(* PLC project H2-1.0.02.project, CODESYS CODESYS V3.5 SP21 Patch 1 *)
(* stored: creationDateTime 2025-11-10T13:44:26.7492399, modificationDateTime 2025-11-05T06:53:28.9174298 *)

{attribute 'qualified_only'}
{attribute 'to_string'}
TYPE Duplex_Mapping : (Z100 := 0, Z201, Z202, TK201, Duplex_End);
END_TYPE

{attribute 'qualified_only'}
{attribute 'to_string'}
TYPE ME44DO_Mapping : (GW202_S4 := 0, GW201_S3, ME44DO_End);
END_TYPE

{attribute 'qualified_only'}
{attribute 'to_string'}
TYPE mPump_Mapping : (mPump_001 := 0, mPump_End);
END_TYPE

{attribute 'qualified_only'}
{attribute 'to_string'}
TYPE s8228_Mapping : (CT_122 := 0, CT_131, CT_142, s8228_End);
END_TYPE

{attribute 'qualified_only'}
{attribute 'to_string'}
TYPE DI_Mapping : (External_Pump_Status := 0, DC_OK, Z201_DC_OK, Spare_3, DI_End);
END_TYPE

{attribute 'qualified_only'}
{attribute 'to_string'}
TYPE Analog_Pump_Mapping : (Analog_Pump_001 := 0, Analog_Pump_End);
END_TYPE

(* values of LS_Mapping: LSLL_101: Z100; LSLL_202: Z201; LSHH_206: Z202-Filter 204A; LSHH_207: Z202-Filter 204B; LSHH_208: Z202-Filter 205A; LSHH_209: Z202-Filter 205B; LSHH_201: EP101; LSHH_204: TK201, *)

{attribute 'qualified_only'}
{attribute 'to_string'}
TYPE LS_Mapping : (LSLL_101 := 0, LSLL_202, LSHH_206, LSLL_210, LSHH_207, LSLL_211, LSHH_208, LSLL_212, LSHH_209, LSLL_213, LSHH_201, LSHH_204, LSLL_203, LSLL_205, LS_End);
END_TYPE

(* values of FIT_Mapping: FT01: FIT_111:=0, FIT_121, *)

{attribute 'qualified_only'}
{attribute 'to_string'}
TYPE FIT_Mapping : (FT01, FIT_End);
END_TYPE

{attribute 'qualified_only'}
{attribute 'to_string'}
TYPE Adam_6217_Mapping : (Adam_6217_001 := 0, Adam_6217_End);
END_TYPE

{attribute 'qualified_only'}
{attribute 'to_string'}
TYPE Adam_6250_Mapping : (Adam_6250_001 := 1, Adam_6250_002, Adam_End);
END_TYPE

(* values of s8098_Mapping: FT_101: Z100; FT_201: Z201; FT_202: Z202; FT_203: TK201 *)

{attribute 'qualified_only'}
{attribute 'to_string'}
TYPE s8098_Mapping : (FT_101 := 0, FT_201, FT_202, FT_204, FT_203, s8098_end);
END_TYPE

(* values of ME44AI_Mapping: GW201_S2: 2; GW201_S4: 4 *)

(* {attribute 'strict'} *)
{attribute 'qualified_only'}
{attribute 'to_string'}
TYPE ME44AI_Mapping : (GW100_S2 := 0, GW100_S3, GW201_S2, GW202_S3, GW201_S4, ME44_AI_End);
END_TYPE

(* values of VFD_Mapping: VFD_101A: VFD-101; VFD_201: Z201; VFD_202: Z202; VFD_102A: EP101; VFD_203: TK201 *)

{attribute 'qualified_only'}
{attribute 'to_string'}
TYPE VFD_Mapping : (VFD_101A := 0, VFD_101B, VFD_201, VFD_201B, VFD_202, VFD_202B, VFD_102A, VFD_102B, VFD_102C, VFD_102D, VFD_102E, VFD_102F, VFD_102G, VFD_102H, VFD_203, VFD_End);
END_TYPE

{attribute 'qualified_only'}
{attribute 'to_string'}
TYPE b8653_mapping : (enum_member := 0, b8653_End);
END_TYPE

(* values of BCV_Mapping: BCV_211: Z202-Filter 204A; BCV_212: Z202-Filter 204B; BCV_217: Z202-Filter 205A; BCV_218: Z202-Filter 205B *)

{attribute 'qualified_only'}
{attribute 'to_string'}
TYPE BCV_Mapping : (BCV_211, BCV_220, BCV_212, BCV_221, BCV_217, BCV_222, BCV_218, BCV_223, BCV_END);
END_TYPE

{attribute 'qualified_only'}
{attribute 'to_string'}
TYPE me64_Mapping : (ME64_001 := 0, ME64_End);
END_TYPE

(* values of Do_Mapping: Stack_R: 5; Skid_201_PWR: 9 *)

{attribute 'qualified_only'}
{attribute 'to_string'}
TYPE Do_Mapping : (Filters_204A := 0, Filters_204B, Filters_205A, Filters_205B, FilterSkid, Stack_R, Stack_Y, Stack_G, Stack_H, Skid_201_PWR, Skid_203_PWR, TK201_PWR_1, TK201_PWR_2, TK201_PWR_3, Do_End);
END_TYPE

(* 8312 Temperature *)
{attribute 'qualified_only'}
{attribute 'to_string'}
TYPE s8412_Mapping : (s8412_001 := 0, s8412_End);
END_TYPE

(* values of s3363_Mapping: ACV_101: Z100; ACV_201: Z201; ACV_207: 3; ACV_208: 5; ACV_213: 7; ACV_214: 9; ACV_219: Z202; ACV_203: TK201 *)

(* {attribute 'strict'} *)
{attribute 'qualified_only'}
{attribute 'to_string'}
TYPE s3363_Mapping : (ACV_101 := 0, ACV_102, ACV_201, ACV_207, ACV_209, ACV_208, ACV_210, ACV_213, ACV_215, ACV_214, ACV_216, ACV_219, ACV_203, ACV_206, ACV_224, ACV_225, ACV_226, s3363_END);
END_TYPE

(* values of s8312_Mapping: PT_101: Z100; PT_201: Z201; PT_202: Z202; PT_203: TK201 *)

(* 8312 Pressure *)
{attribute 'qualified_only'}
{attribute 'to_string'}
TYPE s8312_Mapping : (PT_101 := 0, PT_201, PT_202, PT_204, PT_205, PT_203, S8312_End);
END_TYPE

{attribute 'qualified_only'}
{attribute 'to_string'}
TYPE ME44AO_Mapping : (ME44AO := 0, ME44AO_End);
END_TYPE

{attribute 'qualified_only'}
{attribute 'to_string'}
TYPE Stack_Light_Mapping : (Stack_Light_001 := 0, Stack_Light_End);
END_TYPE

(* values of Line_Mapping: Line_End: Line_3, Line_4, *)

{attribute 'qualified_only'}
{attribute 'to_string'}
TYPE Line_Mapping : (Water := 0, Bleach, Line_End);
END_TYPE

(* values of s8050_Mapping: FT_201A: Z201; FT_202A: Z202; FT_203A: TK201 *)

{attribute 'qualified_only'}
{attribute 'to_string'}
TYPE s8050_Mapping : (FT_201A := 0, FT_202A, FT_204A, FT_203A, s8050_End);
END_TYPE

{attribute 'qualified_only'}
{attribute 'to_string'}
TYPE TT_Mapping : (TT_Start := 0, TT_End);
END_TYPE

(* values of PID_Mapping: Z201_EP101_Level: 3; Z202_Flow: 6; Z202_TK201_Level: 8; TK201_Flow: 11 *)

{attribute 'qualified_only'}
{attribute 'to_string'}
TYPE PID_Mapping : (Z100_Flow := 0, Z100_Pressure, Z100_Level, Z201_EP101_Level, Z201_TK201_Level, Z201_Flow, Z202_Flow, Z202_Pressure, Z202_TK201_Level, Z202_EP101_Level, Z202_Filter_Flow, TK201_Flow, TK201_Pressure, Z202_Recovery_Level, PID_End);
END_TYPE

{attribute 'qualified_only'}
{attribute 'to_string'}
TYPE SV_Mapping : (SV_001 := 0, SV_END);
END_TYPE

(* values of AIT_Mapping: LT_101_P: EP101; LT_202: TK201; LT_202A: 5; LT_01A: 7 *)

{attribute 'qualified_only'}
{attribute 'to_string'}
TYPE AIT_Mapping : (LT_101_P := 0, LT_101_T, LT_201, LT_201A_P, LT_201A_T, LT_202, LT_202A, LT_01A, LT_01B, FT_01, UV_001, AIT_End);
END_TYPE

{attribute 'qualified_only'}
{attribute 'to_string'}
TYPE ACV_Mapping : (ACV_111 := 0, ACV_121, ACV_End);
END_TYPE

(* values of s8605_Mapping: SV_211: Z202-Filter 204A; SV_212: Z202-Filter 204B; SV_217: Z202-Filter 205A; SV_218: Z202-Filter 204A *)

{attribute 'qualified_only'}
{attribute 'to_string'}
TYPE s8605_Mapping : (SV_211 := 0, SV_220, SV_212, SV_221, SV_217, SV_222, SV_218, SV_223, s8605_End);
END_TYPE

{attribute 'qualified_only'}
{attribute 'to_string'}
TYPE ME44DI_Mapping : (GW100_S1 := 0, GW201_S1, GW202_S1, GW202_S2, Me44DI_End);
END_TYPE

PROGRAM Z201_Manager
  VAR
    Local_Status : eZ201_Status;
    tStatus : eZ201_Status;
    Local_Task : eZ201_Task;
    tAlarm : Burkert.Alarm_Window;
    LT201_tAlarm : Burkert.Alarm_Window;
    FT201_Ave : REAL;
    FT201_Gav : REAL;
    FT201_Hav : REAL;
    FT201_Ave_Index : INT;
    Array_Size : UINT;
    VFD_Min_PCT : REAL := 20;
    Level_ton : ton;
  END_VAR
  VAR  (* added by the conversion: wires and edge detectors of the diagram *)
    _SEL3_OUT : ANY;
    _SEL3_OUT_2 : ANY;
    _OR5_OUT : BOOL;
    _SEL21_OUT : ANY;
    _SEL35_OUT : ANY;
    _MAX51_OUT : ANY;
    _LIMIT47_OUT : REAL;
    _GT62_OUT : BOOL;
    _SEL75_OUT : REAL;
    _GT86_OUT : BOOL;
  END_VAR

            PVL.Z201_Config.Mode.eMode:=Burkert.eHOA_Modes.Manual;

Aux();
Alarms();

PVL.Z201_Config.StrMode:=Burkert.Burkert_OSCAT_BASIC.REPLACE_ALL(str:=TO_STRING(PVL.Z201_Config.Mode.eMode) , src:='_' , rep:=' ' );
PVL.Z201_Config.StrStatus:=Burkert.Burkert_OSCAT_BASIC.REPLACE_ALL(str:=TO_STRING(PVL.Z201_Config.Status.eStatus) , src:='_' , rep:=' ' );
PVl.Z201_Config.StrTask:=Burkert.Burkert_OSCAT_BASIC.REPLACE_ALL(str:=TO_STRING(PVL.Z201_Config.Task.eTask) , src:='_' , rep:=' ' );




CASE PVL.Z201_Config.Mode.eMode OF
	Burkert.eHOA_Modes.Off:PVL.Z201_Config.Task.eTask:=eZ201_task.Off;
	//Burkert.eHOA_Modes.Auto:
	//Burkert.eHOA_Modes.Manual:
END_CASE;

CASE pvl.Z201_Config.Task.eTask OF
	eZ201_Task.Off:Task_Off();
	eZ201_Task.Flow:Task_Flow();
	eZ201_Task.TK201_Level:TK201_level();
	eZ201_task.EP101_Level:EP101_Level();
	eZ201_Task.Z100_Flow:Z100_Flow();
	eZ201_Task.Z202_Flow:Z202_Flow();
	eZ201_Task.Drain:Drain();	
	eZ201_Task.Agitate_only:Task_Agitate();
END_CASE





PID_ctrl();
ACV_ctrl();
VFD_ctrl();



          

ACTION Task_Flow:
                IF PVL.Z201_Config.Task.eTask<> Local_Task THEN
	Local_Task:=PVL.Z201_Config.Task.eTask;
	Local_Status:=eZ201_Status.Fixed_Flow_Rate_Transfer_Active;
END_IF;






PVL.PID[PID_Mapping.Z201_Flow].PLC_Target:=PVL.Z201_Config.Target_Flow.Target;


	
	


CASE PVL.Z201_Config.Status.eStatus OF
	
	eZ201_Status.PT201_High_Pressure_Alarm:		Local_Status:=PVL.Z201_Config.Status.eStatus;
	eZ201_Status.PT201_Low_Pressure_Alarm:		Local_Status:=PVL.Z201_Config.Status.eStatus;
	eZ201_Status.FT201_Low_Low_Flow_Alarm:		Local_Status:=PVL.Z201_Config.Status.eStatus;
	//eZ201_Status.LT101_High_High_Alarm:			Local_Status:=PVL.Z201_Config.Status.eStatus;
	//eZ201_Status.LT101_Low_Low_Alarm:			Local_Status:=PVL.Z201_Config.Status.eStatus;
	//eZ201_Status.LT201_High_High_Alarm:			Local_Status:=PVL.Z201_Config.Status.eStatus;
	//eZ201_Status.LT201_Low_Low_Alarm:			Local_Status:=PVL.Z201_Config.Status.eStatus;
	//eZ201_Status.LT201A_High_High_Alarm:		Local_Status:=PVL.Z201_Config.Status.eStatus;
	//eZ201_Status.LT201A_Low_Low_Alarm:			Local_Status:=PVL.Z201_Config.Status.eStatus;
	eZ201_Status.TK201_LSHH204_High_High_Level_Alarm:	Local_Status:=PVL.Z201_Config.Status.eStatus;
	eZ201_Status.Pump_Intake_Dry_LSLL202:		Local_Status:=PVL.Z201_Config.Status.eStatus;
	//eZ201_Status.PT201_High_Pressure_Alarm:		Local_Status:=PVL.Z201_Config.Status.eStatus;
	///eZ201_Status.PT201_Low_Pressure_Alarm:		Local_Status:=PVL.Z201_Config.Status.eStatus;
	//eZ201_Status.FT201_Low_Low_Flow_Alarm:		Local_Status:=PVL.Z201_Config.Status.eStatus;
	
	eZ201_Status.LT201_Low_Low_Alarm:		IF Level_ton.Q THEN local_Status:= eZ201_Status.Waiting_For_Level_OK_LT201; END_IF;
	eZ201_Status.LT202_High_High_Alarm:		IF Level_ton.Q THEN local_Status:= eZ201_Status.Waiting_For_Level_OK_LT202; END_IF;
	eZ201_Status.Waiting_For_Level_OK_LT201:	IF PVL.AIT[AIT_Mapping.LT_201].Status.eStatus=Burkert.eSensor_Status.OK THEN Local_Task:=999; END_IF;
	eZ201_Status.Waiting_For_Level_OK_LT202:	IF PVL.AIT[AIT_Mapping.LT_202].Status.eStatus=Burkert.eSensor_Status.OK THEN Local_Task:=999; END_IF;
	
	eZ201_Status.LT202A_High_High_Alarm:			Local_Status:=eZ201_Status.Waiting_For_Level_OK_LT202a;
	eZ201_Status.Waiting_For_Level_OK_LT202a	:	IF PVL.AIT[ait_mapping.LT_101_P].Status.eStatus=Burkert.eSensor_Status.OK THEN local_Task:=99; END_IF;
	
	

END_CASE;

Evaluate_Task_Flow();
              
END_ACTION

ACTION Z202_Flow:
                IF PVL.Z201_Config.Task.eTask<> Local_Task THEN
	Local_Task:=PVL.Z201_Config.Task.eTask;
END_IF;

Local_Status:=eZ201_Status.Z202_Rate_Match_Transfer_Active;




PVL.PID[PID_Mapping.Z201_Flow].PLC_Target:=PVL.s8098[s8098_Mapping.FT_203].PDO.VolumeFlow.EU;



Evaluate_Z202_Flow();

CASE PVL.Z201_Config.Status.eStatus OF
	//eZ201_Status.LT101_High_High_Alarm:			Local_Status:=PVL.Z201_Config.Status.eStatus;
	//eZ201_Status.LT101_Low_Low_Alarm:			Local_Status:=PVL.Z201_Config.Status.eStatus;
	//eZ201_Status.LT201_High_High_Alarm:			Local_Status:=PVL.Z201_Config.Status.eStatus;
	//eZ201_Status.LT201_Low_Low_Alarm:			Local_Status:=PVL.Z201_Config.Status.eStatus;
	//eZ201_Status.LT201A_High_High_Alarm:		Local_Status:=PVL.Z201_Config.Status.eStatus;
	//eZ201_Status.LT201A_Low_Low_Alarm:			Local_Status:=PVL.Z201_Config.Status.eStatus;
	eZ201_Status.TK201_LSHH204_High_High_Level_Alarm:	Local_Status:=PVL.Z201_Config.Status.eStatus;
	eZ201_Status.Pump_Intake_Dry_LSLL202:		Local_Status:=PVL.Z201_Config.Status.eStatus;
	eZ201_Status.PT201_High_Pressure_Alarm:		Local_Status:=PVL.Z201_Config.Status.eStatus;
	///eZ201_Status.PT201_Low_Pressure_Alarm:		Local_Status:=PVL.Z201_Config.Status.eStatus;
	eZ201_Status.FT201_Low_Low_Flow_Alarm:		Local_Status:=PVL.Z201_Config.Status.eStatus;
	eZ201_Status.LT201_Low_Low_Alarm:		IF Level_ton.Q THEN local_Status:= eZ201_Status.Waiting_For_Level_OK_LT201; END_IF;
	eZ201_Status.LT202_High_High_Alarm:		IF Level_ton.Q THEN local_Status:= eZ201_Status.Waiting_For_Level_OK_LT202; END_IF;
	eZ201_Status.Waiting_For_Level_OK_LT201:	IF PVL.AIT[AIT_Mapping.LT_201].Status.eStatus=Burkert.eSensor_Status.OK THEN Local_Task:=999; END_IF;
	eZ201_Status.Waiting_For_Level_OK_LT202:	IF PVL.AIT[AIT_Mapping.LT_202].Status.eStatus=Burkert.eSensor_Status.OK THEN Local_Task:=999; END_IF;
	eZ201_Status.LT202A_High_High_Alarm:			Local_Status:=eZ201_Status.Waiting_For_Level_OK_LT202a;
	eZ201_Status.Waiting_For_Level_OK_LT202a	:	IF PVL.AIT[ait_mapping.LT_101_P].Status.eStatus=Burkert.eSensor_Status.OK THEN local_Task:=99; END_IF;
	

	eZ201_Status.PT201_Low_Pressure_Alarm:		Local_Status:=PVL.Z201_Config.Status.eStatus;
	//eZ201_Status.FT201_Low_Low_Flow_Alarm:		Local_Status:=PVL.Z201_Config.Status.eStatus;

END_CASE
              
END_ACTION

ACTION Task_OFF:
                IF PVL.Z201_Config.Task.eTask<> Local_Task THEN
	Local_Task:=PVL.Z201_Config.Task.eTask;
END_IF;

Local_Status:=eZ201_Status.Off;

Evaluate_Off();

              
END_ACTION

ACTION Drain:
                IF PVL.Z201_Config.Task.eTask<> Local_Task THEN
	Local_Task:=PVL.Z201_Config.Task.eTask;
	Local_Status:=eZ201_Status.Drain_Active;
END_IF;






PVL.PID[PID_Mapping.Z201_Flow].PLC_Target:=PVl.Z201_Config.Drain_Rate.Target;



Evaluate_Drain();


CASE PVL.Z201_Config.Status.eStatus OF
	//eZ201_Status.LT101_High_High_Alarm:			Local_Status:=PVL.Z201_Config.Status.eStatus;
	//eZ201_Status.LT101_Low_Low_Alarm:			Local_Status:=PVL.Z201_Config.Status.eStatus;
	//eZ201_Status.LT201_High_High_Alarm:			Local_Status:=PVL.Z201_Config.Status.eStatus;
	//eZ201_Status.LT201_Low_Low_Alarm:			Local_Status:=PVL.Z201_Config.Status.eStatus;
	//eZ201_Status.LT201A_High_High_Alarm:		Local_Status:=PVL.Z201_Config.Status.eStatus;
	//eZ201_Status.LT201A_Low_Low_Alarm:			Local_Status:=PVL.Z201_Config.Status.eStatus;
	//eZ201_Status.TK201_High_High_Level_Alarm:	Local_Status:=PVL.Z201_Config.Status.eStatus;
	eZ201_Status.Pump_Intake_Dry_LSLL202:		Local_Status:=PVL.Z201_Config.Status.eStatus;
	eZ201_Status.Drain_Complete:				Local_Status:=PVL.Z201_Config.Status.eStatus;
	
	eZ201_Status.PT201_High_Pressure_Alarm:		Local_Status:=eZ201_Status.PT201_High_Pressure_Alarm;
	eZ201_Status.PT201_Low_Pressure_Alarm:		Local_Status:=eZ201_Status.PT201_Low_Pressure_Alarm;
	eZ201_Status.FT201_Low_Low_Flow_Alarm:		Local_Status:=eZ201_Status.FT201_Low_Low_Flow_Alarm;
	
	eZ201_Status.LT201_Low_Low_Alarm:		IF Level_ton.Q THEN local_Status:= eZ201_Status.Waiting_For_Level_OK_LT201; END_IF;
	eZ201_Status.LT202_High_High_Alarm:		IF Level_ton.Q THEN local_Status:= eZ201_Status.Waiting_For_Level_OK_LT202; END_IF;
	eZ201_Status.Waiting_For_Level_OK_LT201:	IF PVL.AIT[AIT_Mapping.LT_201].Status.eStatus=Burkert.eSensor_Status.OK THEN Local_Task:=999; END_IF;
	eZ201_Status.Waiting_For_Level_OK_LT202:	IF PVL.AIT[AIT_Mapping.LT_202].Status.eStatus=Burkert.eSensor_Status.OK THEN Local_Task:=999; END_IF;
	
	eZ201_Status.LT202A_High_High_Alarm:			Local_Status:=eZ201_Status.Waiting_For_Level_OK_LT202a;
	eZ201_Status.Waiting_For_Level_OK_LT202a	:	IF PVL.AIT[ait_mapping.LT_101_P].Status.eStatus=Burkert.eSensor_Status.OK THEN local_Task:=99; END_IF;
	

END_CASE;
              
END_ACTION

ACTION Evaluate_Off:
                tStatus:=Local_Status;

IF GVl.LS[LS_Mapping.LSLL_202].Status.eStatus=Burkert.DI_Status.No_Liquid_Detected_Alarm THEN tStatus:=eZ201_Status.Pump_Intake_Dry_LSLL202; END_IF;
IF GVl.LS[LS_Mapping.LSHH_204 ].Status.eStatus=Burkert.DI_Status.Liquid_Detected_Alarm THEN tStatus:=eZ201_Status.TK201_LSHH204_High_High_Level_Alarm; END_IF;

//IF NOT(Network.VFD[VFD_Mapping.VFD_102A].Ready) THEN tStatus:=eZ201_Status.VFD_102A_Not_Ready;	END_IF;
//IF NOT(Network.VFD[VFD_Mapping.VFD_102B].Ready) THEN tStatus:=eZ201_Status.VFD_102B_Not_Ready;	END_IF;
//IF NOT(Network.VFD[VFD_Mapping.VFD_102C].Ready) THEN tStatus:=eZ201_Status.VFD_102C_Not_Ready;	END_IF;
//IF NOT(Network.VFD[VFD_Mapping.VFD_102D].Ready) THEN tStatus:=eZ201_Status.VFD_102D_Not_Ready;	END_IF;
//IF NOT(Network.VFD[VFD_Mapping.VFD_102E].Ready) THEN tStatus:=eZ201_Status.VFD_102E_Not_Ready;	END_IF;
//IF NOT(Network.VFD[VFD_Mapping.VFD_102F].Ready) THEN tStatus:=eZ201_Status.VFD_102F_Not_Ready;	END_IF;
//IF NOT(Network.VFD[VFD_Mapping.VFD_102G].Ready) THEN tStatus:=eZ201_Status.VFD_102G_Not_Ready;	END_IF;
//IF NOT(Network.VFD[VFD_Mapping.VFD_102H].Ready) THEN tStatus:=eZ201_Status.VFD_102H_Not_Ready;	END_IF;

IF Network.VFD[VFD_Mapping.VFD_102A].Status=Burkert.eVFD_Status.High_High_Current_Alarm THEN tStatus:=eZ201_Status.VFD_102A_High_Current;	END_IF;
IF Network.VFD[VFD_Mapping.VFD_102B].Status=Burkert.eVFD_Status.High_High_Current_Alarm THEN tStatus:=eZ201_Status.VFD_102B_High_Current;	END_IF;
IF Network.VFD[VFD_Mapping.VFD_102C].Status=Burkert.eVFD_Status.High_High_Current_Alarm THEN tStatus:=eZ201_Status.VFD_102C_High_Current;	END_IF;
IF Network.VFD[VFD_Mapping.VFD_102D].Status=Burkert.eVFD_Status.High_High_Current_Alarm THEN tStatus:=eZ201_Status.VFD_102D_High_Current;	END_IF;
//IF Network.VFD[VFD_Mapping.VFD_102E].Status=Burkert.eVFD_Status.High_High_Current_Alarm THEN tStatus:=eZ201_Status.VFD_102E_High_Current;	END_IF;
//IF Network.VFD[VFD_Mapping.VFD_102F].Status=Burkert.eVFD_Status.High_High_Current_Alarm THEN tStatus:=eZ201_Status.VFD_102F_High_Current;	END_IF;
//IF Network.VFD[VFD_Mapping.VFD_102G].Status=Burkert.eVFD_Status.High_High_Current_Alarm THEN tStatus:=eZ201_Status.VFD_102G_High_Current;	END_IF;
//IF Network.VFD[VFD_Mapping.VFD_102H].Status=Burkert.eVFD_Status.High_High_Current_Alarm THEN tStatus:=eZ201_Status.VFD_102H_High_Current;	END_IF;


IF NOT(Network.VFD[VFD_Mapping.VFD_201].Ready) THEN tStatus:=eZ201_Status.VFD_201_Not_Ready;	END_IF;

IF NOT(GVL.s3363[s3363_mapping.ACV_201].Ready) THEN	tStatus:=eZ201_Status.ACV_201_Not_Ready;	END_IF;
	
IF NOT(PVl.s8312[s8312_mapping.PT_201].Ready) THEN	tStatus:=eZ201_status.PT201_Not_Ready;	END_IF;
IF NOT(PVL.s8098[s8098_Mapping.FT_201].Ready) THEN	tStatus:=eZ201_status.FT201_Not_Ready;	END_IF;


IF NOT(PVL.AIT[AIT_Mapping.LT_101_P].Ready) THEN tStatus:=eZ201_Status.LT101_Not_Ready;	END_IF;
IF NOT(PVL.AIT[AIT_Mapping.LT_201A_P].Ready) THEN tStatus:=eZ201_Status.LT201A_Not_Ready;	END_IF;
IF NOT(PVL.AIT[AIT_Mapping.LT_201].Ready) THEN tStatus:=eZ201_Status.LT201_Not_Ready;	END_IF;

IF PVL.AIT[AIT_Mapping.LT_101_P].Status.eStatus=Burkert.eSensor_Status.HiHi_Alarm THEN	tStatus:=eZ201_Status.LT101_High_High_Alarm; END_IF;
IF PVL.AIT[AIT_Mapping.LT_101_P].Status.eStatus=Burkert.eSensor_Status.Low_Low_Alarm THEN	tStatus:=eZ201_Status.LT101_Low_Low_Alarm; END_IF;

IF PVL.AIT[AIT_Mapping.LT_201A_P].Status.eStatus=Burkert.eSensor_Status.HiHi_Alarm THEN	tStatus:=eZ201_Status.LT201A_High_High_Alarm; END_IF;
IF PVL.AIT[AIT_Mapping.LT_201A_P].Status.eStatus=Burkert.eSensor_Status.Low_Low_Alarm THEN	tStatus:=eZ201_Status.LT201A_Low_Low_Alarm; END_IF;

IF PVL.AIT[AIT_Mapping.LT_201].Status.eStatus=Burkert.eSensor_Status.HiHi_Alarm THEN	tStatus:=eZ201_Status.LT201_High_High_Alarm; END_IF;
IF PVL.AIT[AIT_Mapping.LT_201].Status.eStatus=Burkert.eSensor_Status.Low_Low_Alarm THEN	tStatus:=eZ201_Status.LT201_Low_Low_Alarm; END_IF;


PVL.Z201_Config.Status.eStatus:=tStatus;

              
END_ACTION

ACTION Z100_Flow:
                IF PVL.Z201_Config.Task.eTask<> Local_Task THEN
	Local_Task:=PVL.Z201_Config.Task.eTask;
END_IF;

Local_Status:=eZ201_Status.Z100_Rate_Match_Transfer_Active;




PVL.PID[PID_Mapping.Z201_Flow].PLC_Target:=PVL.s8098[s8098_Mapping.FT_101].PDO.VolumeFlow.EU;




Evaluate_Z100_Flow();

CASE PVL.Z201_Config.Status.eStatus OF
	//eZ201_Status.LT101_High_High_Alarm:			Local_Status:=PVL.Z201_Config.Status.eStatus;
	//eZ201_Status.LT101_Low_Low_Alarm:			Local_Status:=PVL.Z201_Config.Status.eStatus;
	//eZ201_Status.LT201_High_High_Alarm:			Local_Status:=PVL.Z201_Config.Status.eStatus;
	//eZ201_Status.LT201_Low_Low_Alarm:			Local_Status:=PVL.Z201_Config.Status.eStatus;
	//eZ201_Status.LT201A_High_High_Alarm:		Local_Status:=PVL.Z201_Config.Status.eStatus;
	//eZ201_Status.LT201A_Low_Low_Alarm:			Local_Status:=PVL.Z201_Config.Status.eStatus;
	eZ201_Status.TK201_LSHH204_High_High_Level_Alarm:	Local_Status:=PVL.Z201_Config.Status.eStatus;
	eZ201_Status.Pump_Intake_Dry_LSLL202:		Local_Status:=PVL.Z201_Config.Status.eStatus;
	eZ201_Status.PT201_High_Pressure_Alarm:		Local_Status:=PVL.Z201_Config.Status.eStatus;
	///eZ201_Status.PT201_Low_Pressure_Alarm:		Local_Status:=PVL.Z201_Config.Status.eStatus;
	eZ201_Status.FT201_Low_Low_Flow_Alarm:		Local_Status:=PVL.Z201_Config.Status.eStatus;
	
	eZ201_Status.LT201_Low_Low_Alarm:		IF Level_ton.Q THEN local_Status:= eZ201_Status.Waiting_For_Level_OK_LT201; END_IF;
	eZ201_Status.LT202_High_High_Alarm:		IF Level_ton.Q THEN local_Status:= eZ201_Status.Waiting_For_Level_OK_LT202; END_IF;
	eZ201_Status.Waiting_For_Level_OK_LT201:	IF PVL.AIT[AIT_Mapping.LT_201].Status.eStatus=Burkert.eSensor_Status.OK THEN Local_Task:=999; END_IF;
	eZ201_Status.Waiting_For_Level_OK_LT202:	IF PVL.AIT[AIT_Mapping.LT_202].Status.eStatus=Burkert.eSensor_Status.OK THEN Local_Task:=999; END_IF;
	eZ201_Status.LT202A_High_High_Alarm:			Local_Status:=eZ201_Status.Waiting_For_Level_OK_LT202a;
	eZ201_Status.Waiting_For_Level_OK_LT202a	:	IF PVL.AIT[ait_mapping.LT_101_P].Status.eStatus=Burkert.eSensor_Status.OK THEN local_Task:=99; END_IF;
	
	//eZ201_Status.PT201_High_Pressure_Alarm:		Local_Status:=PVL.Z201_Config.Status.eStatus;
	eZ201_Status.PT201_Low_Pressure_Alarm:		Local_Status:=PVL.Z201_Config.Status.eStatus;
	//eZ201_Status.FT201_Low_Low_Flow_Alarm:		Local_Status:=PVL.Z201_Config.Status.eStatus;

END_CASE
              
END_ACTION

ACTION ACV_ctrl:
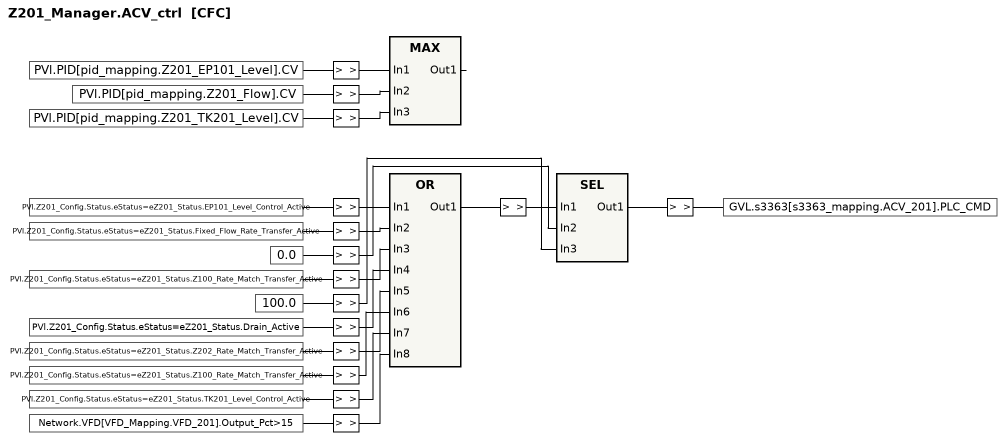
(* CFC diagram, written out as Structured Text *)
GVL.s3363[s3363_mapping.ACV_201].PLC_CMD := _SEL3_OUT;
_SEL3_OUT := SEL((PVl.Z201_Config.Status.eStatus=eZ201_Status.EP101_Level_Control_Active) OR (PVl.Z201_Config.Status.eStatus=eZ201_Status.Fixed_Flow_Rate_Transfer_Active) OR (PVl.Z201_Config.Status.eStatus=eZ201_Status.Z100_Rate_Match_Transfer_Active) OR (PVl.Z201_Config.Status.eStatus=eZ201_Status.Drain_Active) OR (PVl.Z201_Config.Status.eStatus=eZ201_Status.Z202_Rate_Match_Transfer_Active) OR (PVl.Z201_Config.Status.eStatus=eZ201_Status.Z100_Rate_Match_Transfer_Active) OR (PVl.Z201_Config.Status.eStatus=eZ201_Status.TK201_Level_Control_Active) OR (Network.VFD[VFD_Mapping.VFD_201].Output_Pct>15), 0.0, 100.0);
MAX(PVl.PID[pid_mapping.Z201_EP101_Level].CV, PVl.PID[pid_mapping.Z201_Flow].CV, PVl.PID[pid_mapping.Z201_TK201_Level].CV);
END_ACTION

ACTION Evaluate_Z100_Flow:
                tStatus:=Local_Status;

IF GVl.LS[LS_Mapping.LSLL_202].Status.eStatus=Burkert.DI_Status.No_Liquid_Detected_Alarm THEN tStatus:=eZ201_Status.Pump_Intake_Dry_LSLL202; END_IF;
IF GVl.LS[LS_Mapping.LSHH_204 ].Status.eStatus=Burkert.DI_Status.Liquid_Detected_Alarm THEN tStatus:=eZ201_Status.TK201_LSHH204_High_High_Level_Alarm; END_IF;

//IF NOT(Network.VFD[VFD_Mapping.VFD_102A].Ready) THEN tStatus:=eZ201_Status.VFD_102A_Not_Ready;	END_IF;
//IF NOT(Network.VFD[VFD_Mapping.VFD_102B].Ready) THEN tStatus:=eZ201_Status.VFD_102B_Not_Ready;	END_IF;
//IF NOT(Network.VFD[VFD_Mapping.VFD_102C].Ready) THEN tStatus:=eZ201_Status.VFD_102C_Not_Ready;	END_IF;
//IF NOT(Network.VFD[VFD_Mapping.VFD_102D].Ready) THEN tStatus:=eZ201_Status.VFD_102D_Not_Ready;	END_IF;
//IF NOT(Network.VFD[VFD_Mapping.VFD_102E].Ready) THEN tStatus:=eZ201_Status.VFD_102E_Not_Ready;	END_IF;
//IF NOT(Network.VFD[VFD_Mapping.VFD_102F].Ready) THEN tStatus:=eZ201_Status.VFD_102F_Not_Ready;	END_IF;
//IF NOT(Network.VFD[VFD_Mapping.VFD_102G].Ready) THEN tStatus:=eZ201_Status.VFD_102G_Not_Ready;	END_IF;
//IF NOT(Network.VFD[VFD_Mapping.VFD_102H].Ready) THEN tStatus:=eZ201_Status.VFD_102H_Not_Ready;	END_IF;
IF NOT(Network.VFD[VFD_Mapping.VFD_201].Ready) THEN tStatus:=eZ201_Status.VFD_201_Not_Ready;	END_IF;

//IF Network.VFD[VFD_Mapping.VFD_102A].Status=Burkert.eVFD_Status.High_High_Current_Alarm THEN tStatus:=eZ201_Status.VFD_102A_High_Current;	END_IF;
//IF Network.VFD[VFD_Mapping.VFD_102B].Status=Burkert.eVFD_Status.High_High_Current_Alarm THEN tStatus:=eZ201_Status.VFD_102B_High_Current;	END_IF;
//IF Network.VFD[VFD_Mapping.VFD_102C].Status=Burkert.eVFD_Status.High_High_Current_Alarm THEN tStatus:=eZ201_Status.VFD_102C_High_Current;	END_IF;
//IF Network.VFD[VFD_Mapping.VFD_102D].Status=Burkert.eVFD_Status.High_High_Current_Alarm THEN tStatus:=eZ201_Status.VFD_102D_High_Current;	END_IF;
//IF Network.VFD[VFD_Mapping.VFD_102E].Status=Burkert.eVFD_Status.High_High_Current_Alarm THEN tStatus:=eZ201_Status.VFD_102E_High_Current;	END_IF;
//IF Network.VFD[VFD_Mapping.VFD_102F].Status=Burkert.eVFD_Status.High_High_Current_Alarm THEN tStatus:=eZ201_Status.VFD_102F_High_Current;	END_IF;
//IF Network.VFD[VFD_Mapping.VFD_102G].Status=Burkert.eVFD_Status.High_High_Current_Alarm THEN tStatus:=eZ201_Status.VFD_102G_High_Current;	END_IF;
//IF Network.VFD[VFD_Mapping.VFD_102H].Status=Burkert.eVFD_Status.High_High_Current_Alarm THEN tStatus:=eZ201_Status.VFD_102H_High_Current;	END_IF;



IF NOT(GVL.s3363[s3363_mapping.ACV_201].Ready) THEN	tStatus:=eZ201_Status.ACV_201_Not_Ready;	END_IF;
	
IF NOT(PVl.s8312[s8312_mapping.PT_201].Ready) THEN	tStatus:=eZ201_status.PT201_Not_Ready;	END_IF;
IF PVL.s8312[s8312_Mapping.PT_201].Status.eStatus=Burkert.eSensor_Status.HiHi_Alarm THEN tStatus:=eZ201_Status.PT201_High_Pressure_Alarm; END_IF;
//IF PVL.s8312[s8312_Mapping.PT_201].Status.eStatus=Burkert.eSensor_Status.Low_Low_Alarm THEN tStatus:=eZ201_Status.PT201_Low_Pressure_Alarm; END_IF;

IF NOT(PVL.s8098[s8098_Mapping.FT_201].Ready) THEN	tStatus:=eZ201_status.FT201_Not_Ready;	END_IF;
IF PVL.s8098[s8098_Mapping.FT_201].PDO.VolumeFlow.Status.eStatus=Burkert.eSensor_Status.Low_Low_Alarm THEN tStatus:=eZ201_status.FT201_Low_Low_Flow_Alarm;	END_IF;


//IF NOT(PVL.AIT[AIT_Mapping.LT_101_P].Ready) THEN tStatus:=eZ201_Status.LT101_Not_Ready;	END_IF;
//IF NOT(PVL.AIT[AIT_Mapping.LT_201A_P].Ready) THEN tStatus:=eZ201_Status.LT201A_Not_Ready;	END_IF;
IF NOT(PVL.AIT[AIT_Mapping.LT_201].Ready) THEN tStatus:=eZ201_Status.LT201_Not_Ready;	END_IF;
IF NOT(PVL.AIT[AIT_Mapping.LT_202].Ready) THEN tStatus:=eZ201_Status.LT202_Not_Ready;	END_IF;
//IF NOT(PVL.AIT[AIT_Mapping.LT_202a].Ready) THEN tStatus:=eZ201_Status.LT202a_Not_Ready;	END_IF;

//IF PVL.AIT[AIT_Mapping.LT_101_P].Status.eStatus=Burkert.eSensor_Status.HiHi_Alarm THEN	tStatus:=eZ201_Status.LT101_High_High_Alarm; END_IF;
///IF PVL.AIT[AIT_Mapping.LT_101_P].Status.eStatus=Burkert.eSensor_Status.Low_Low_Alarm THEN	tStatus:=eZ201_Status.LT101_Low_Low_Alarm; END_IF;

//IF PVL.AIT[AIT_Mapping.LT_201A_P].Status.eStatus=Burkert.eSensor_Status.HiHi_Alarm THEN	tStatus:=eZ201_Status.LT201A_High_High_Alarm; END_IF;
//IF PVL.AIT[AIT_Mapping.LT_201A_P].Status.eStatus=Burkert.eSensor_Status.Low_Low_Alarm THEN	tStatus:=eZ201_Status.LT201A_Low_Low_Alarm; END_IF;

//IF PVL.AIT[AIT_Mapping.LT_201].Status.eStatus=Burkert.eSensor_Status.HiHi_Alarm THEN	tStatus:=eZ201_Status.LT201_High_High_Alarm; END_IF;
IF PVL.AIT[AIT_Mapping.LT_201].Status.eStatus=Burkert.eSensor_Status.Low_Low_Alarm THEN	tStatus:=eZ201_Status.LT201_Low_Low_Alarm; END_IF;
//IF PVL.AIT[AIT_Mapping.LT_202].Status.eStatus=Burkert.eSensor_Status.HiHi_Alarm THEN	tStatus:=eZ201_Status.LT202_High_High_Alarm; END_IF;
IF PVL.AIT[AIT_Mapping.LT_202a].Status.eStatus=Burkert.eSensor_Status.HiHi_Alarm THEN	tStatus:=eZ201_Status.LT202a_High_High_Alarm; END_IF;


IF PVl.s8312[s8312_mapping.PT_201].Status.eStatus=Burkert.eSensor_Status.Low_Low_Alarm 					THEN	tStatus:=eZ201_Status.PT201_Low_Pressure_Alarm; END_IF;
IF PVl.s8312[s8312_mapping.PT_201].Status.eStatus=Burkert.eSensor_Status.HiHi_Alarm 					THEN	tStatus:=eZ201_Status.PT201_High_Pressure_Alarm; END_IF;
IF PVL.s8098[s8098_Mapping.FT_201].PDO.VolumeFlow.Status.eStatus=Burkert.eSensor_Status.Low_Low_Alarm	THEN	tStatus:=ez201_Status.FT201_Low_Low_Flow_Alarm; END_IF;


PVL.Z201_Config.Status.eStatus:=tStatus;

              
END_ACTION

ACTION TK201_Level:
                IF PVL.Z201_Config.Task.eTask<> Local_Task THEN
	Local_Task:=PVL.Z201_Config.Task.eTask;
	Local_Status:=eZ201_Status.TK201_Level_Control_Active;
END_IF;





PVL.PID[PID_Mapping.Z201_TK201_Level ].PLC_Target:=PVL.Z201_Config.Target_TK201_Level.Target;


(*
PVL.AIT[ait_Mapping.LT_101_P].Alarm_Config:=PVL.AIT[AIT_Mapping.LT_201].Alarm_Config;

*)
CASE PVL.Z201_Config.Status.eStatus OF
	//eZ201_Status.LT101_High_High_Alarm:			Local_Status:=PVL.Z201_Config.Status.eStatus;
	//eZ201_Status.LT101_Low_Low_Alarm:			Local_Status:=PVL.Z201_Config.Status.eStatus;
	//eZ201_Status.LT201_High_High_Alarm:			Local_Status:=PVL.Z201_Config.Status.eStatus;
	//eZ201_Status.LT201_Low_Low_Alarm:			Local_Status:=PVL.Z201_Config.Status.eStatus;
	//eZ201_Status.LT201A_High_High_Alarm:		Local_Status:=PVL.Z201_Config.Status.eStatus;
	//eZ201_Status.LT201A_Low_Low_Alarm:			Local_Status:=PVL.Z201_Config.Status.eStatus;
	eZ201_Status.TK201_LSHH204_High_High_Level_Alarm:	Local_Status:=PVL.Z201_Config.Status.eStatus;
	eZ201_Status.Pump_Intake_Dry_LSLL202:		Local_Status:=PVL.Z201_Config.Status.eStatus;
	eZ201_Status.PT201_High_Pressure_Alarm:		Local_Status:=PVL.Z201_Config.Status.eStatus;
	///eZ201_Status.PT201_Low_Pressure_Alarm:		Local_Status:=PVL.Z201_Config.Status.eStatus;
	eZ201_Status.FT201_Low_Low_Flow_Alarm:		Local_Status:=PVL.Z201_Config.Status.eStatus;
	
	eZ201_Status.LT201_Low_Low_Alarm:		IF Level_ton.Q THEN local_Status:= eZ201_Status.Waiting_For_Level_OK_LT201; END_IF;
	eZ201_Status.LT202_High_High_Alarm:		IF Level_ton.Q THEN local_Status:= eZ201_Status.Waiting_For_Level_OK_LT202; END_IF;
	eZ201_Status.Waiting_For_Level_OK_LT201:	IF PVL.AIT[AIT_Mapping.LT_201].Status.eStatus=Burkert.eSensor_Status.OK THEN Local_Task:=999; END_IF;
	eZ201_Status.Waiting_For_Level_OK_LT202:	IF PVL.AIT[AIT_Mapping.LT_202].Status.eStatus=Burkert.eSensor_Status.OK THEN Local_Task:=999; END_IF;
	
	eZ201_Status.LT202A_High_High_Alarm:			Local_Status:=eZ201_Status.Waiting_For_Level_OK_LT202a;
	eZ201_Status.Waiting_For_Level_OK_LT202a	:	IF PVL.AIT[ait_mapping.LT_101_P].Status.eStatus=Burkert.eSensor_Status.OK THEN local_Task:=99; END_IF;
	
	//eZ201_Status.PT201_High_Pressure_Alarm:		Local_Status:=PVL.Z201_Config.Status.eStatus;
	eZ201_Status.PT201_Low_Pressure_Alarm:		Local_Status:=PVL.Z201_Config.Status.eStatus;
	//eZ201_Status.FT201_Low_Low_Flow_Alarm:		Local_Status:=PVL.Z201_Config.Status.eStatus;

END_CASE;

Evaluate_TK201_Level();
              
END_ACTION

ACTION VFD_ctrl:
(* CFC diagram, written out as Structured Text *)
Network.VFD[VFD_Mapping.VFD_102B].PLC_CMD := _SEL3_OUT_2;
_SEL3_OUT_2 := SEL(_OR5_OUT, PVL.Z201_Config.Mixer_Target[1], 0.0);
Network.VFD[VFD_Mapping.VFD_102B].PLC_Run := _SEL3_OUT_2 > 5;
Network.VFD[VFD_Mapping.VFD_102C].PLC_CMD := _SEL21_OUT;
_SEL21_OUT := SEL(_OR5_OUT, PVL.Z201_Config.Mixer_Target[2], 0.0);
Network.VFD[VFD_Mapping.VFD_102C].PLC_Run := _SEL21_OUT > 5;
Network.VFD[VFD_Mapping.VFD_102D].PLC_CMD := _SEL35_OUT;
_SEL35_OUT := SEL(_OR5_OUT, PVL.Z201_Config.Mixer_Target[3], 0.0);
Network.VFD[VFD_Mapping.VFD_102D].PLC_Run := _SEL35_OUT > 5;
_LIMIT47_OUT := LIMIT(0.0, _MAX51_OUT, 100.0);
_MAX51_OUT := MAX(PVl.PID[pid_mapping.Z201_EP101_Level].CV, PVl.PID[pid_mapping.Z201_Flow].CV, PVl.PID[pid_mapping.Z201_TK201_Level].CV);
Network.VFD[VFD_Mapping.VFD_201].PLC_CMD := _LIMIT47_OUT;
_GT62_OUT := _LIMIT47_OUT > 5;
Network.VFD[VFD_Mapping.VFD_201].PLC_Run := _GT62_OUT AND True AND NOT (PVL.Z201_Config.Task.eTask=eZ201_Task.Off);
_SEL75_OUT := SEL(_OR5_OUT, PVL.Z201_Config.Mixer_Target[0], 0.0);
Network.VFD[VFD_Mapping.VFD_102A].PLC_CMD := _SEL75_OUT;
Network.VFD[VFD_Mapping.VFD_102A].PLC_Run := _GT86_OUT;
_GT86_OUT := _SEL75_OUT > 5;
_OR5_OUT := (PVL.Z201_Config.Task.eTask=eZ201_Task.Off) OR (PVL.Z201_Config.Task.eTask=eZ201_Task.Drain);
(* drawn but not wired to any output: GVL.s3363[s3363_mapping.ACV_201].PDO.Pos, GVL.s3363[s3363_mapping.ACV_201].Mode.eMode=Burkert.eACV_Modes.Auto *)
END_ACTION

ACTION Evaluate_Drain:
                tStatus:=Local_Status;

IF GVl.LS[LS_Mapping.LSLL_202].Status.eStatus=Burkert.DI_Status.No_Liquid_Detected_Alarm THEN tStatus:=eZ201_Status.Drain_Complete; END_IF;
IF GVl.LS[LS_Mapping.LSHH_204 ].Status.eStatus=Burkert.DI_Status.Liquid_Detected_Alarm THEN tStatus:=eZ201_Status.TK201_LSHH204_High_High_Level_Alarm; END_IF;

//IF NOT(Network.VFD[VFD_Mapping.VFD_102A].Ready) THEN tStatus:=eZ201_Status.VFD_102A_Not_Ready;	END_IF;
//IF NOT(Network.VFD[VFD_Mapping.VFD_102B].Ready) THEN tStatus:=eZ201_Status.VFD_102B_Not_Ready;	END_IF;
//IF NOT(Network.VFD[VFD_Mapping.VFD_102C].Ready) THEN tStatus:=eZ201_Status.VFD_102C_Not_Ready;	END_IF;
//IF NOT(Network.VFD[VFD_Mapping.VFD_102D].Ready) THEN tStatus:=eZ201_Status.VFD_102D_Not_Ready;	END_IF;
//IF NOT(Network.VFD[VFD_Mapping.VFD_102E].Ready) THEN tStatus:=eZ201_Status.VFD_102E_Not_Ready;	END_IF;
//IF NOT(Network.VFD[VFD_Mapping.VFD_102F].Ready) THEN tStatus:=eZ201_Status.VFD_102F_Not_Ready;	END_IF;
//IF NOT(Network.VFD[VFD_Mapping.VFD_102G].Ready) THEN tStatus:=eZ201_Status.VFD_102G_Not_Ready;	END_IF;
//IF NOT(Network.VFD[VFD_Mapping.VFD_102H].Ready) THEN tStatus:=eZ201_Status.VFD_102H_Not_Ready;	END_IF;
IF NOT(Network.VFD[VFD_Mapping.VFD_201].Ready) THEN tStatus:=eZ201_Status.VFD_201_Not_Ready;	END_IF;

IF NOT(GVL.s3363[s3363_mapping.ACV_201].Ready) THEN	tStatus:=eZ201_Status.ACV_201_Not_Ready;	END_IF;
	
IF NOT(PVl.s8312[s8312_mapping.PT_201].Ready) THEN	tStatus:=eZ201_status.PT201_Not_Ready;	END_IF;
IF NOT(PVL.s8098[s8098_Mapping.FT_201].Ready) THEN	tStatus:=eZ201_status.FT201_Not_Ready;	END_IF;


//IF NOT(PVL.AIT[AIT_Mapping.LT_101_P].Ready) THEN tStatus:=eZ201_Status.LT101_Not_Ready;	END_IF;
//IF NOT(PVL.AIT[AIT_Mapping.LT_201A_P].Ready) THEN tStatus:=eZ201_Status.LT201A_Not_Ready;	END_IF;
IF NOT(PVL.AIT[AIT_Mapping.LT_201].Ready) THEN tStatus:=eZ201_Status.LT201_Not_Ready;	END_IF;

//IF PVL.AIT[AIT_Mapping.LT_101_P].Status.eStatus=Burkert.eSensor_Status.HiHi_Alarm THEN	tStatus:=eZ201_Status.LT101_High_High_Alarm; END_IF;
//IF PVL.AIT[AIT_Mapping.LT_101_P].Status.eStatus=Burkert.eSensor_Status.Low_Low_Alarm THEN	tStatus:=eZ201_Status.LT101_Low_Low_Alarm; END_IF;

//IF PVL.AIT[AIT_Mapping.LT_201A_P].Status.eStatus=Burkert.eSensor_Status.HiHi_Alarm THEN	tStatus:=eZ201_Status.LT201A_High_High_Alarm; END_IF;
//IF PVL.AIT[AIT_Mapping.LT_201A_P].Status.eStatus=Burkert.eSensor_Status.Low_Low_Alarm THEN	tStatus:=eZ201_Status.LT201A_Low_Low_Alarm; END_IF;

///IF PVL.AIT[AIT_Mapping.LT_201].Status.eStatus=Burkert.eSensor_Status.HiHi_Alarm THEN	tStatus:=eZ201_Status.LT201_High_High_Alarm; END_IF;
//IF PVL.AIT[AIT_Mapping.LT_201].Status.eStatus=Burkert.eSensor_Status.Low_Low_Alarm THEN	tStatus:=eZ201_Status.LT201_Low_Low_Alarm; END_IF;


IF PVl.s8312[s8312_mapping.PT_201].Status.eStatus=Burkert.eSensor_Status.Low_Low_Alarm 					THEN	tStatus:=eZ201_Status.PT201_Low_Pressure_Alarm; END_IF;
IF PVl.s8312[s8312_mapping.PT_201].Status.eStatus=Burkert.eSensor_Status.HiHi_Alarm 					THEN	tStatus:=eZ201_Status.PT201_High_Pressure_Alarm; END_IF;
IF PVL.s8098[s8098_Mapping.FT_201].PDO.VolumeFlow.Status.eStatus=Burkert.eSensor_Status.Low_Low_Alarm	THEN	tStatus:=ez201_Status.FT201_Low_Low_Flow_Alarm; END_IF;

IF PVL.AIT[AIT_Mapping.LT_202a].Status.eStatus=Burkert.eSensor_Status.HiHi_Alarm THEN	tStatus:=eZ201_Status.LT202a_High_High_Alarm; END_IF;

PVL.Z201_Config.Status.eStatus:=tStatus;

              
END_ACTION

ACTION PID_ctrl:
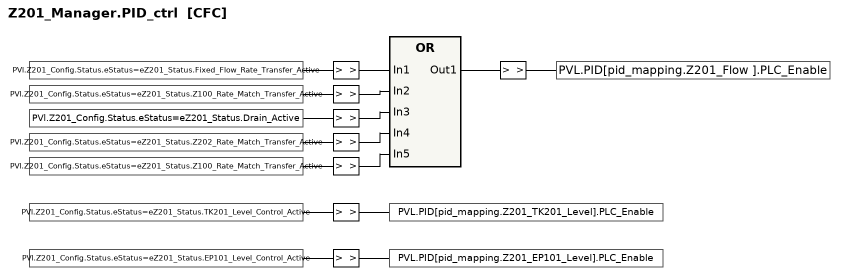
(* CFC diagram, written out as Structured Text *)
PVL.PID[pid_mapping.Z201_Flow ].PLC_Enable := (PVl.Z201_Config.Status.eStatus=eZ201_Status.Fixed_Flow_Rate_Transfer_Active) OR (PVl.Z201_Config.Status.eStatus=eZ201_Status.Z100_Rate_Match_Transfer_Active) OR (PVl.Z201_Config.Status.eStatus=eZ201_Status.Drain_Active) OR (PVl.Z201_Config.Status.eStatus=eZ201_Status.Z202_Rate_Match_Transfer_Active) OR (PVl.Z201_Config.Status.eStatus=eZ201_Status.Z100_Rate_Match_Transfer_Active);
PVL.PID[pid_mapping.Z201_TK201_Level].PLC_Enable := PVl.Z201_Config.Status.eStatus=eZ201_Status.TK201_Level_Control_Active;
PVL.PID[pid_mapping.Z201_EP101_Level].PLC_Enable := PVl.Z201_Config.Status.eStatus=eZ201_Status.EP101_Level_Control_Active;
END_ACTION

ACTION Evaluate_TK201_level:
                tStatus:=Local_Status;

IF GVl.LS[LS_Mapping.LSLL_202].Status.eStatus=Burkert.DI_Status.No_Liquid_Detected_Alarm THEN tStatus:=eZ201_Status.Pump_Intake_Dry_LSLL202; END_IF;
IF GVl.LS[LS_Mapping.LSHH_204 ].Status.eStatus=Burkert.DI_Status.Liquid_Detected_Alarm THEN tStatus:=eZ201_Status.TK201_LSHH204_High_High_Level_Alarm; END_IF;

//IF NOT(Network.VFD[VFD_Mapping.VFD_102A].Ready) THEN tStatus:=eZ201_Status.VFD_102A_Not_Ready;	END_IF;
//IF NOT(Network.VFD[VFD_Mapping.VFD_102B].Ready) THEN tStatus:=eZ201_Status.VFD_102B_Not_Ready;	END_IF;
//IF NOT(Network.VFD[VFD_Mapping.VFD_102C].Ready) THEN tStatus:=eZ201_Status.VFD_102C_Not_Ready;	END_IF;
//IF NOT(Network.VFD[VFD_Mapping.VFD_102D].Ready) THEN tStatus:=eZ201_Status.VFD_102D_Not_Ready;	END_IF;
//IF NOT(Network.VFD[VFD_Mapping.VFD_102E].Ready) THEN tStatus:=eZ201_Status.VFD_102E_Not_Ready;	END_IF;
//IF NOT(Network.VFD[VFD_Mapping.VFD_102F].Ready) THEN tStatus:=eZ201_Status.VFD_102F_Not_Ready;	END_IF;
//IF NOT(Network.VFD[VFD_Mapping.VFD_102G].Ready) THEN tStatus:=eZ201_Status.VFD_102G_Not_Ready;	END_IF;
//IF NOT(Network.VFD[VFD_Mapping.VFD_102H].Ready) THEN tStatus:=eZ201_Status.VFD_102H_Not_Ready;	END_IF;
IF NOT(Network.VFD[VFD_Mapping.VFD_201].Ready) THEN tStatus:=eZ201_Status.VFD_201_Not_Ready;	END_IF;

//IF Network.VFD[VFD_Mapping.VFD_102A].Status=Burkert.eVFD_Status.High_High_Current_Alarm THEN tStatus:=eZ201_Status.VFD_102A_High_Current;	END_IF;
//IF Network.VFD[VFD_Mapping.VFD_102B].Status=Burkert.eVFD_Status.High_High_Current_Alarm THEN tStatus:=eZ201_Status.VFD_102B_High_Current;	END_IF;
//IF Network.VFD[VFD_Mapping.VFD_102C].Status=Burkert.eVFD_Status.High_High_Current_Alarm THEN tStatus:=eZ201_Status.VFD_102C_High_Current;	END_IF;
//IF Network.VFD[VFD_Mapping.VFD_102D].Status=Burkert.eVFD_Status.High_High_Current_Alarm THEN tStatus:=eZ201_Status.VFD_102D_High_Current;	END_IF;
//IF Network.VFD[VFD_Mapping.VFD_102E].Status=Burkert.eVFD_Status.High_High_Current_Alarm THEN tStatus:=eZ201_Status.VFD_102E_High_Current;	END_IF;
//IF Network.VFD[VFD_Mapping.VFD_102F].Status=Burkert.eVFD_Status.High_High_Current_Alarm THEN tStatus:=eZ201_Status.VFD_102F_High_Current;	END_IF;
//IF Network.VFD[VFD_Mapping.VFD_102G].Status=Burkert.eVFD_Status.High_High_Current_Alarm THEN tStatus:=eZ201_Status.VFD_102G_High_Current;	END_IF;
//IF Network.VFD[VFD_Mapping.VFD_102H].Status=Burkert.eVFD_Status.High_High_Current_Alarm THEN tStatus:=eZ201_Status.VFD_102H_High_Current;	END_IF;


IF NOT(GVL.s3363[s3363_mapping.ACV_201].Ready) THEN	tStatus:=eZ201_Status.ACV_201_Not_Ready;	END_IF;
	
IF NOT(PVl.s8312[s8312_mapping.PT_201].Ready) THEN	tStatus:=eZ201_status.PT201_Not_Ready;	END_IF;
IF PVL.s8312[s8312_Mapping.PT_201].Status.eStatus=Burkert.eSensor_Status.HiHi_Alarm THEN tStatus:=eZ201_Status.PT201_High_Pressure_Alarm; END_IF;
//IF PVL.s8312[s8312_Mapping.PT_201].Status.eStatus=Burkert.eSensor_Status.Low_Low_Alarm THEN tStatus:=eZ201_Status.PT201_Low_Pressure_Alarm; END_IF;

IF NOT(PVL.s8098[s8098_Mapping.FT_201].Ready) THEN	tStatus:=eZ201_status.FT201_Not_Ready;	END_IF;
IF PVL.s8098[s8098_Mapping.FT_201].PDO.VolumeFlow.Status.eStatus=Burkert.eSensor_Status.Low_Low_Alarm THEN tStatus:=eZ201_status.FT201_Low_Low_Flow_Alarm;	END_IF;


//IF NOT(PVL.AIT[AIT_Mapping.LT_101_P].Ready) THEN tStatus:=eZ201_Status.LT101_Not_Ready;	END_IF;
//IF NOT(PVL.AIT[AIT_Mapping.LT_201A_P].Ready) THEN tStatus:=eZ201_Status.LT201A_Not_Ready;	END_IF;
IF NOT(PVL.AIT[AIT_Mapping.LT_201].Ready) THEN tStatus:=eZ201_Status.LT201_Not_Ready;	END_IF;
IF NOT(PVL.AIT[AIT_Mapping.LT_202].Ready) THEN tStatus:=eZ201_Status.LT202_Not_Ready;	END_IF;
//IF NOT(PVL.AIT[AIT_Mapping.LT_202a].Ready) THEN tStatus:=eZ201_Status.LT202a_Not_Ready;	END_IF;

//IF PVL.AIT[AIT_Mapping.LT_101_P].Status.eStatus=Burkert.eSensor_Status.HiHi_Alarm THEN	tStatus:=eZ201_Status.LT101_High_High_Alarm; END_IF;
///IF PVL.AIT[AIT_Mapping.LT_101_P].Status.eStatus=Burkert.eSensor_Status.Low_Low_Alarm THEN	tStatus:=eZ201_Status.LT101_Low_Low_Alarm; END_IF;

//IF PVL.AIT[AIT_Mapping.LT_201A_P].Status.eStatus=Burkert.eSensor_Status.HiHi_Alarm THEN	tStatus:=eZ201_Status.LT201A_High_High_Alarm; END_IF;
//IF PVL.AIT[AIT_Mapping.LT_201A_P].Status.eStatus=Burkert.eSensor_Status.Low_Low_Alarm THEN	tStatus:=eZ201_Status.LT201A_Low_Low_Alarm; END_IF;

//IF PVL.AIT[AIT_Mapping.LT_201].Status.eStatus=Burkert.eSensor_Status.HiHi_Alarm THEN	tStatus:=eZ201_Status.LT201_High_High_Alarm; END_IF;
IF PVL.AIT[AIT_Mapping.LT_201].Status.eStatus=Burkert.eSensor_Status.Low_Low_Alarm THEN	tStatus:=eZ201_Status.LT201_Low_Low_Alarm; END_IF;
//IF PVL.AIT[AIT_Mapping.LT_202].Status.eStatus=Burkert.eSensor_Status.HiHi_Alarm THEN	tStatus:=eZ201_Status.LT202_High_High_Alarm; END_IF;
///IF PVL.AIT[AIT_Mapping.LT_202a].Status.eStatus=Burkert.eSensor_Status.HiHi_Alarm THEN	tStatus:=eZ201_Status.LT202a_High_High_Alarm; END_IF;

IF PVl.s8312[s8312_mapping.PT_201].Status.eStatus=Burkert.eSensor_Status.Low_Low_Alarm 					THEN	tStatus:=eZ201_Status.PT201_Low_Pressure_Alarm; END_IF;
IF PVl.s8312[s8312_mapping.PT_201].Status.eStatus=Burkert.eSensor_Status.HiHi_Alarm 					THEN	tStatus:=eZ201_Status.PT201_High_Pressure_Alarm; END_IF;
//IF PVL.s8098[s8098_Mapping.FT_201].PDO.VolumeFlow.Status.eStatus=Burkert.eSensor_Status.Low_Low_Alarm	THEN	tStatus:=ez201_Status.FT201_Low_Low_Flow_Alarm; END_IF;

PVL.Z201_Config.Status.eStatus:=tStatus;

              
END_ACTION

ACTION EP101_Level:
                IF PVL.Z201_Config.Task.eTask<> Local_Task THEN
	Local_Task:=PVL.Z201_Config.Task.eTask;
	Local_Status:=eZ201_Status.EP101_Level_Control_Active;
END_IF;






PVL.PID[PID_Mapping.Z201_EP101_Level].PLC_Target:=PVL.Z201_Config.Target_EP101_Level.Target;




Evaluate_EP101_Level();

CASE PVL.Z201_Config.Status.eStatus OF
	//eZ201_Status.LT101_High_High_Alarm:			Local_Status:=PVL.Z201_Config.Status.eStatus;
	//eZ201_Status.LT101_Low_Low_Alarm:			Local_Status:=PVL.Z201_Config.Status.eStatus;
	//eZ201_Status.LT201_High_High_Alarm:			Local_Status:=PVL.Z201_Config.Status.eStatus;
	//eZ201_Status.LT201_Low_Low_Alarm:			Local_Status:=PVL.Z201_Config.Status.eStatus;
	//eZ201_Status.LT201A_High_High_Alarm:		Local_Status:=PVL.Z201_Config.Status.eStatus;
	//eZ201_Status.LT201A_Low_Low_Alarm:			Local_Status:=PVL.Z201_Config.Status.eStatus;
	eZ201_Status.TK201_LSHH204_High_High_Level_Alarm:	Local_Status:=PVL.Z201_Config.Status.eStatus;
	eZ201_Status.Pump_Intake_Dry_LSLL202:		Local_Status:=PVL.Z201_Config.Status.eStatus;
	eZ201_Status.PT201_High_Pressure_Alarm:		Local_Status:=PVL.Z201_Config.Status.eStatus;
	///eZ201_Status.PT201_Low_Pressure_Alarm:		Local_Status:=PVL.Z201_Config.Status.eStatus;
	eZ201_Status.FT201_Low_Low_Flow_Alarm:		Local_Status:=PVL.Z201_Config.Status.eStatus;
	
	eZ201_Status.LT201_Low_Low_Alarm:		IF Level_ton.Q THEN local_Status:= eZ201_Status.Waiting_For_Level_OK_LT201; END_IF;
	eZ201_Status.LT202_High_High_Alarm:		IF Level_ton.Q THEN local_Status:= eZ201_Status.Waiting_For_Level_OK_LT202; END_IF;
	eZ201_Status.Waiting_For_Level_OK_LT201:	IF PVL.AIT[AIT_Mapping.LT_201].Status.eStatus=Burkert.eSensor_Status.OK THEN Local_Task:=999; END_IF;
	eZ201_Status.Waiting_For_Level_OK_LT202:	IF PVL.AIT[AIT_Mapping.LT_202].Status.eStatus=Burkert.eSensor_Status.OK THEN Local_Task:=999; END_IF;
	
	

	eZ201_Status.PT201_Low_Pressure_Alarm:		Local_Status:=PVL.Z201_Config.Status.eStatus;
END_CASE;
              
END_ACTION

ACTION Evaluate_Z202_Flow:
                tStatus:=Local_Status;

IF GVl.LS[LS_Mapping.LSLL_202].Status.eStatus=Burkert.DI_Status.No_Liquid_Detected_Alarm THEN tStatus:=eZ201_Status.Pump_Intake_Dry_LSLL202; END_IF;
IF GVl.LS[LS_Mapping.LSHH_204 ].Status.eStatus=Burkert.DI_Status.Liquid_Detected_Alarm THEN tStatus:=eZ201_Status.TK201_LSHH204_High_High_Level_Alarm; END_IF;

//IF NOT(Network.VFD[VFD_Mapping.VFD_102A].Ready) THEN tStatus:=eZ201_Status.VFD_102A_Not_Ready;	END_IF;
//IF NOT(Network.VFD[VFD_Mapping.VFD_102B].Ready) THEN tStatus:=eZ201_Status.VFD_102B_Not_Ready;	END_IF;
//IF NOT(Network.VFD[VFD_Mapping.VFD_102C].Ready) THEN tStatus:=eZ201_Status.VFD_102C_Not_Ready;	END_IF;
//IF NOT(Network.VFD[VFD_Mapping.VFD_102D].Ready) THEN tStatus:=eZ201_Status.VFD_102D_Not_Ready;	END_IF;
//IF NOT(Network.VFD[VFD_Mapping.VFD_102E].Ready) THEN tStatus:=eZ201_Status.VFD_102E_Not_Ready;	END_IF;
//IF NOT(Network.VFD[VFD_Mapping.VFD_102F].Ready) THEN tStatus:=eZ201_Status.VFD_102F_Not_Ready;	END_IF;
//IF NOT(Network.VFD[VFD_Mapping.VFD_102G].Ready) THEN tStatus:=eZ201_Status.VFD_102G_Not_Ready;	END_IF;
//IF NOT(Network.VFD[VFD_Mapping.VFD_102H].Ready) THEN tStatus:=eZ201_Status.VFD_102H_Not_Ready;	END_IF;
IF NOT(Network.VFD[VFD_Mapping.VFD_201].Ready) THEN tStatus:=eZ201_Status.VFD_201_Not_Ready;	END_IF;

//IF Network.VFD[VFD_Mapping.VFD_102A].Status=Burkert.eVFD_Status.High_High_Current_Alarm THEN tStatus:=eZ201_Status.VFD_102A_High_Current;	END_IF;
//IF Network.VFD[VFD_Mapping.VFD_102B].Status=Burkert.eVFD_Status.High_High_Current_Alarm THEN tStatus:=eZ201_Status.VFD_102B_High_Current;	END_IF;
//IF Network.VFD[VFD_Mapping.VFD_102C].Status=Burkert.eVFD_Status.High_High_Current_Alarm THEN tStatus:=eZ201_Status.VFD_102C_High_Current;	END_IF;
//IF Network.VFD[VFD_Mapping.VFD_102D].Status=Burkert.eVFD_Status.High_High_Current_Alarm THEN tStatus:=eZ201_Status.VFD_102D_High_Current;	END_IF;
//IF Network.VFD[VFD_Mapping.VFD_102E].Status=Burkert.eVFD_Status.High_High_Current_Alarm THEN tStatus:=eZ201_Status.VFD_102E_High_Current;	END_IF;
//IF Network.VFD[VFD_Mapping.VFD_102F].Status=Burkert.eVFD_Status.High_High_Current_Alarm THEN tStatus:=eZ201_Status.VFD_102F_High_Current;	END_IF;
//IF Network.VFD[VFD_Mapping.VFD_102G].Status=Burkert.eVFD_Status.High_High_Current_Alarm THEN tStatus:=eZ201_Status.VFD_102G_High_Current;	END_IF;
//IF Network.VFD[VFD_Mapping.VFD_102H].Status=Burkert.eVFD_Status.High_High_Current_Alarm THEN tStatus:=eZ201_Status.VFD_102H_High_Current;	END_IF;



IF NOT(GVL.s3363[s3363_mapping.ACV_201].Ready) THEN	tStatus:=eZ201_Status.ACV_201_Not_Ready;	END_IF;
	
IF NOT(PVl.s8312[s8312_mapping.PT_201].Ready) THEN	tStatus:=eZ201_status.PT201_Not_Ready;	END_IF;
IF PVL.s8312[s8312_Mapping.PT_201].Status.eStatus=Burkert.eSensor_Status.HiHi_Alarm THEN tStatus:=eZ201_Status.PT201_High_Pressure_Alarm; END_IF;
//IF PVL.s8312[s8312_Mapping.PT_201].Status.eStatus=Burkert.eSensor_Status.Low_Low_Alarm THEN tStatus:=eZ201_Status.PT201_Low_Pressure_Alarm; END_IF;

IF NOT(PVL.s8098[s8098_Mapping.FT_201].Ready) THEN	tStatus:=eZ201_status.FT201_Not_Ready;	END_IF;
IF PVL.s8098[s8098_Mapping.FT_201].PDO.VolumeFlow.Status.eStatus=Burkert.eSensor_Status.Low_Low_Alarm THEN tStatus:=eZ201_status.FT201_Low_Low_Flow_Alarm;	END_IF;


//IF NOT(PVL.AIT[AIT_Mapping.LT_101_P].Ready) THEN tStatus:=eZ201_Status.LT101_Not_Ready;	END_IF;
//IF NOT(PVL.AIT[AIT_Mapping.LT_201A_P].Ready) THEN tStatus:=eZ201_Status.LT201A_Not_Ready;	END_IF;
IF NOT(PVL.AIT[AIT_Mapping.LT_201].Ready) THEN tStatus:=eZ201_Status.LT201_Not_Ready;	END_IF;
IF NOT(PVL.AIT[AIT_Mapping.LT_202].Ready) THEN tStatus:=eZ201_Status.LT202_Not_Ready;	END_IF;
//IF NOT(PVL.AIT[AIT_Mapping.LT_202a].Ready) THEN tStatus:=eZ201_Status.LT202a_Not_Ready;	END_IF;

//IF PVL.AIT[AIT_Mapping.LT_101_P].Status.eStatus=Burkert.eSensor_Status.HiHi_Alarm THEN	tStatus:=eZ201_Status.LT101_High_High_Alarm; END_IF;
///IF PVL.AIT[AIT_Mapping.LT_101_P].Status.eStatus=Burkert.eSensor_Status.Low_Low_Alarm THEN	tStatus:=eZ201_Status.LT101_Low_Low_Alarm; END_IF;

//IF PVL.AIT[AIT_Mapping.LT_201A_P].Status.eStatus=Burkert.eSensor_Status.HiHi_Alarm THEN	tStatus:=eZ201_Status.LT201A_High_High_Alarm; END_IF;
//IF PVL.AIT[AIT_Mapping.LT_201A_P].Status.eStatus=Burkert.eSensor_Status.Low_Low_Alarm THEN	tStatus:=eZ201_Status.LT201A_Low_Low_Alarm; END_IF;

//IF PVL.AIT[AIT_Mapping.LT_201].Status.eStatus=Burkert.eSensor_Status.HiHi_Alarm THEN	tStatus:=eZ201_Status.LT201_High_High_Alarm; END_IF;
IF PVL.AIT[AIT_Mapping.LT_201].Status.eStatus=Burkert.eSensor_Status.Low_Low_Alarm THEN	tStatus:=eZ201_Status.LT201_Low_Low_Alarm; END_IF;
//IF PVL.AIT[AIT_Mapping.LT_202].Status.eStatus=Burkert.eSensor_Status.HiHi_Alarm THEN	tStatus:=eZ201_Status.LT202_High_High_Alarm; END_IF;
IF PVL.AIT[AIT_Mapping.LT_202a].Status.eStatus=Burkert.eSensor_Status.HiHi_Alarm THEN	tStatus:=eZ201_Status.LT202a_High_High_Alarm; END_IF;


IF PVl.s8312[s8312_mapping.PT_201].Status.eStatus=Burkert.eSensor_Status.Low_Low_Alarm 					THEN	tStatus:=eZ201_Status.PT201_Low_Pressure_Alarm; END_IF;
IF PVl.s8312[s8312_mapping.PT_201].Status.eStatus=Burkert.eSensor_Status.HiHi_Alarm 					THEN	tStatus:=eZ201_Status.PT201_High_Pressure_Alarm; END_IF;
IF PVL.s8098[s8098_Mapping.FT_201].PDO.VolumeFlow.Status.eStatus=Burkert.eSensor_Status.Low_Low_Alarm	THEN	tStatus:=ez201_Status.FT201_Low_Low_Flow_Alarm; END_IF;


PVL.Z201_Config.Status.eStatus:=tStatus;

              
END_ACTION

ACTION Aux:
                Level_ton(PT:=T#10S, IN:=(
		PVL.Z201_Config.Status.eStatus=eZ201_Status.LT201_Low_Low_Alarm OR 
		PVL.Z201_Config.Status.eStatus=eZ202_Status.LT202_High_High_Alarm OR
		PVL.Z201_Config.Status.eStatus=eZ202_Status.LT202a_High_High_Alarm)
);
PVL.Z201_Config.EP101_Volume_m3:= (PVL.Z201_Config.EP101_Area  * (PVL.AIT[AIT_Mapping.LT_101_P].EU /100));


Array_Size:=SIZEOF(GVl.FT201_Ave);
IF GVL.CLK_500ms THEN
	IF FT201_Ave_Index<50 AND PVL.s8098[s8098_Mapping.FT_201].PDO.VolumeFlow.EU> 0 THEN	
		GVl.FT201_Ave[FT201_Ave_Index]:=PVL.s8098[s8098_Mapping.FT_201].PDO.VolumeFlow.EU;
		FT201_Ave_Index:=FT201_Ave_Index+1;
	ELSE
		Burkert.MEM.MemMove(pSource:= ADR(GVl.FT201_Ave[1]), pDestination:=ADR(GVl.FT201_Ave[0]) , uiNumberOfBytes:=(SIZEOF(GVl.FT201_Ave)-4) );
		GVl.FT201_Ave[49]:=PVL.s8098[s8098_Mapping.FT_201].PDO.VolumeFlow.EU;
	END_IF;

	IF FT201_Ave_Index>0 THEN
		FT201_Ave:=Burkert.Burkert_OSCAT_BASIC.ARRAY_AVG (	pt:=ADR(GVl.FT201_Ave),	size:=SIZEOF(GVl.FT201_Ave));
		//FT201_Gav:=Burkert.Burkert_OSCAT_BASIC.ARRAY_GAV (	pt:=ADR(GVl.FT201_Ave[0]),size:=TO_UINT(FT201_Ave_Index*4));
		FT201_Hav:=Burkert.Burkert_OSCAT_BASIC.ARRAY_HAV (	pt:=ADR(GVl.FT201_Ave[0]),size:=TO_UINT(FT201_Ave_Index*4));
	END_IF;
	
END_IF;

IF FT201_Ave=0 AND Network.VFD[VFD_Mapping.VFD_201].Output_Pct<10 THEN 	FT201_Ave_Index:=0; END_IF;
PVl.PID[pid_mapping.Z201_Flow].Actual:=FT201_AVE;

Network.VFD[VFD_Mapping.VFD_102A].Current_Alarm:=PVL.Z201_Config.Mixer_Motor_Current;
Network.VFD[VFD_Mapping.VFD_102b].Current_Alarm:=PVL.Z201_Config.Mixer_Motor_Current;
Network.VFD[VFD_Mapping.VFD_102c].Current_Alarm:=PVL.Z201_Config.Mixer_Motor_Current;
Network.VFD[VFD_Mapping.VFD_102d].Current_Alarm:=PVL.Z201_Config.Mixer_Motor_Current;
Network.VFD[VFD_Mapping.VFD_102E].Current_Alarm:=PVL.Z201_Config.Mixer_Motor_Current;
Network.VFD[VFD_Mapping.VFD_102F].Current_Alarm:=PVL.Z201_Config.Mixer_Motor_Current;
Network.VFD[VFD_Mapping.VFD_102G].Current_Alarm:=PVL.Z201_Config.Mixer_Motor_Current;
Network.VFD[VFD_Mapping.VFD_102H].Current_Alarm:=PVL.Z201_Config.Mixer_Motor_Current;
              
END_ACTION

ACTION Evaluate_EP101_Level:
                tStatus:=Local_Status;

IF GVl.LS[LS_Mapping.LSLL_202].Status.eStatus=Burkert.DI_Status.No_Liquid_Detected_Alarm THEN tStatus:=eZ201_Status.Pump_Intake_Dry_LSLL202; END_IF;
IF GVl.LS[LS_Mapping.LSHH_204 ].Status.eStatus=Burkert.DI_Status.Liquid_Detected_Alarm THEN tStatus:=eZ201_Status.TK201_LSHH204_High_High_Level_Alarm; END_IF;

//IF NOT(Network.VFD[VFD_Mapping.VFD_102A].Ready) THEN tStatus:=eZ201_Status.VFD_102A_Not_Ready;	END_IF;
//IF NOT(Network.VFD[VFD_Mapping.VFD_102B].Ready) THEN tStatus:=eZ201_Status.VFD_102B_Not_Ready;	END_IF;
//IF NOT(Network.VFD[VFD_Mapping.VFD_102C].Ready) THEN tStatus:=eZ201_Status.VFD_102C_Not_Ready;	END_IF;
//IF NOT(Network.VFD[VFD_Mapping.VFD_102D].Ready) THEN tStatus:=eZ201_Status.VFD_102D_Not_Ready;	END_IF;
//IF NOT(Network.VFD[VFD_Mapping.VFD_102E].Ready) THEN tStatus:=eZ201_Status.VFD_102E_Not_Ready;	END_IF;
//IF NOT(Network.VFD[VFD_Mapping.VFD_102F].Ready) THEN tStatus:=eZ201_Status.VFD_102F_Not_Ready;	END_IF;
//IF NOT(Network.VFD[VFD_Mapping.VFD_102G].Ready) THEN tStatus:=eZ201_Status.VFD_102G_Not_Ready;	END_IF;
//IF NOT(Network.VFD[VFD_Mapping.VFD_102H].Ready) THEN tStatus:=eZ201_Status.VFD_102H_Not_Ready;	END_IF;
IF NOT(Network.VFD[VFD_Mapping.VFD_201].Ready) THEN tStatus:=eZ201_Status.VFD_201_Not_Ready;	END_IF;


//IF Network.VFD[VFD_Mapping.VFD_102A].Status=Burkert.eVFD_Status.High_High_Current_Alarm THEN tStatus:=eZ201_Status.VFD_102A_High_Current;	END_IF;
//IF Network.VFD[VFD_Mapping.VFD_102B].Status=Burkert.eVFD_Status.High_High_Current_Alarm THEN tStatus:=eZ201_Status.VFD_102B_High_Current;	END_IF;
//IF Network.VFD[VFD_Mapping.VFD_102C].Status=Burkert.eVFD_Status.High_High_Current_Alarm THEN tStatus:=eZ201_Status.VFD_102C_High_Current;	END_IF;
//IF Network.VFD[VFD_Mapping.VFD_102D].Status=Burkert.eVFD_Status.High_High_Current_Alarm THEN tStatus:=eZ201_Status.VFD_102D_High_Current;	END_IF;
//IF Network.VFD[VFD_Mapping.VFD_102E].Status=Burkert.eVFD_Status.High_High_Current_Alarm THEN tStatus:=eZ201_Status.VFD_102E_High_Current;	END_IF;
//IF Network.VFD[VFD_Mapping.VFD_102F].Status=Burkert.eVFD_Status.High_High_Current_Alarm THEN tStatus:=eZ201_Status.VFD_102F_High_Current;	END_IF;
//IF Network.VFD[VFD_Mapping.VFD_102G].Status=Burkert.eVFD_Status.High_High_Current_Alarm THEN tStatus:=eZ201_Status.VFD_102G_High_Current;	END_IF;
//IF Network.VFD[VFD_Mapping.VFD_102H].Status=Burkert.eVFD_Status.High_High_Current_Alarm THEN tStatus:=eZ201_Status.VFD_102H_High_Current;	END_IF;


IF NOT(GVL.s3363[s3363_mapping.ACV_201].Ready) THEN	tStatus:=eZ201_Status.ACV_201_Not_Ready;	END_IF;
	
IF NOT(PVl.s8312[s8312_mapping.PT_201].Ready) THEN	tStatus:=eZ201_status.PT201_Not_Ready;	END_IF;
IF NOT(PVL.s8098[s8098_Mapping.FT_201].Ready) THEN	tStatus:=eZ201_status.FT201_Not_Ready;	END_IF;



//IF NOT(PVL.AIT[AIT_Mapping.LT_101_P].Ready) THEN tStatus:=eZ201_Status.LT101_Not_Ready;	END_IF;
//IF NOT(PVL.AIT[AIT_Mapping.LT_201A_P].Ready) THEN tStatus:=eZ201_Status.LT201A_Not_Ready;	END_IF;
IF NOT(PVL.AIT[AIT_Mapping.LT_201].Ready) THEN tStatus:=eZ201_Status.LT201_Not_Ready;	END_IF;
IF NOT(PVL.AIT[AIT_Mapping.LT_202].Ready) THEN tStatus:=eZ201_Status.LT202_Not_Ready;	END_IF;
//IF NOT(PVL.AIT[AIT_Mapping.LT_202a].Ready) THEN tStatus:=eZ201_Status.LT202a_Not_Ready;	END_IF;

//IF PVL.AIT[AIT_Mapping.LT_101_P].Status.eStatus=Burkert.eSensor_Status.HiHi_Alarm THEN	tStatus:=eZ201_Status.LT101_High_High_Alarm; END_IF;
///IF PVL.AIT[AIT_Mapping.LT_101_P].Status.eStatus=Burkert.eSensor_Status.Low_Low_Alarm THEN	tStatus:=eZ201_Status.LT101_Low_Low_Alarm; END_IF;

//IF PVL.AIT[AIT_Mapping.LT_201A_P].Status.eStatus=Burkert.eSensor_Status.HiHi_Alarm THEN	tStatus:=eZ201_Status.LT201A_High_High_Alarm; END_IF;
//IF PVL.AIT[AIT_Mapping.LT_201A_P].Status.eStatus=Burkert.eSensor_Status.Low_Low_Alarm THEN	tStatus:=eZ201_Status.LT201A_Low_Low_Alarm; END_IF;

//IF PVL.AIT[AIT_Mapping.LT_201].Status.eStatus=Burkert.eSensor_Status.HiHi_Alarm THEN	tStatus:=eZ201_Status.LT201_High_High_Alarm; END_IF;
IF PVL.AIT[AIT_Mapping.LT_201].Status.eStatus=Burkert.eSensor_Status.Low_Low_Alarm THEN	tStatus:=eZ201_Status.LT201_Low_Low_Alarm; END_IF;
//IF PVL.AIT[AIT_Mapping.LT_202].Status.eStatus=Burkert.eSensor_Status.HiHi_Alarm THEN	tStatus:=eZ201_Status.LT202_High_High_Alarm; END_IF;
IF PVL.AIT[AIT_Mapping.LT_202a].Status.eStatus=Burkert.eSensor_Status.HiHi_Alarm THEN	tStatus:=eZ201_Status.LT202a_High_High_Alarm; END_IF;


IF PVl.s8312[s8312_mapping.PT_201].Status.eStatus=Burkert.eSensor_Status.Low_Low_Alarm 					THEN	tStatus:=eZ201_Status.PT201_Low_Pressure_Alarm; END_IF;
IF PVl.s8312[s8312_mapping.PT_201].Status.eStatus=Burkert.eSensor_Status.HiHi_Alarm 					THEN	tStatus:=eZ201_Status.PT201_High_Pressure_Alarm; END_IF;
IF PVL.s8098[s8098_Mapping.FT_201].PDO.VolumeFlow.Status.eStatus=Burkert.eSensor_Status.Low_Low_Alarm	THEN	tStatus:=ez201_Status.FT201_Low_Low_Flow_Alarm; END_IF;



PVL.Z201_Config.Status.eStatus:=tStatus;

              
END_ACTION

ACTION Alarms:
                LT201_tAlarm.Target:=PVL.AIT[AIT_mapping.LT_201].Analog_Scale.Eu_Max * (PVL.Z201_Config.Target_EP101_Level.Target/100);
LT201_tAlarm.Warn_Window:=PVL.AIT[AIT_mapping.LT_201].Analog_Scale.Eu_Max * (PVL.Z201_Config.Target_EP101_Level.Warn_Window/100);
LT201_tAlarm.Alarm_Window:=PVL.AIT[AIT_mapping.LT_201].Analog_Scale.Eu_Max * (PVL.Z201_Config.Target_EP101_Level.Alarm_Window/100);
LT201_tAlarm.Alarm_Delay:=PVL.Z201_Config.Target_EP101_Level.Alarm_Delay;
Burkert.Alarm_Window_Convert(window:=LT201_tAlarm,Config:=PVL.AIT[AIT_Mapping.LT_201].Alarm_Config);
PVL.AIT[ait_Mapping.LT_201A_P].Alarm_Config:=PVL.AIT[AIT_Mapping.LT_201].Alarm_Config;
//PVL.AIT[ait_Mapping.LT_101_P].Alarm_Config:=PVL.AIT[AIT_Mapping.LT_201].Alarm_Config;


tAlarm.Target:=PVL.AIT[AIT_mapping.LT_201A_P].Analog_Scale.Eu_Max * (PVL.Z201_Config.Target_EP101_Level.Target/100);
tAlarm.Warn_Window:=PVL.AIT[AIT_mapping.LT_201A_P].Analog_Scale.Eu_Max * (PVL.Z201_Config.Target_EP101_Level.Warn_Window/100);
tAlarm.Alarm_Window:=PVL.AIT[AIT_mapping.LT_201A_P].Analog_Scale.Eu_Max * (PVL.Z201_Config.Target_EP101_Level.Alarm_Window/100);
tAlarm.Alarm_Delay:=PVL.Z201_Config.Target_EP101_Level.Alarm_Delay;
Burkert.Alarm_Window_Convert(window:=tAlarm,Config:=PVL.AIT[AIT_Mapping.LT_201A_P].Alarm_Config);
(*
tAlarm.Target:=PVL.AIT[AIT_mapping.LT_101_P].Analog_Scale.Eu_Max * (PVL.Z201_Config.Target_EP101_Level.Target/100);
tAlarm.Warn_Window:=PVL.AIT[AIT_mapping.LT_101_P].Analog_Scale.Eu_Max * (PVL.Z201_Config.Target_EP101_Level.Warn_Window/100);
tAlarm.Alarm_Window:=PVL.AIT[AIT_mapping.LT_101_P].Analog_Scale.Eu_Max * (PVL.Z201_Config.Target_EP101_Level.Alarm_Window/100);
tAlarm.Alarm_Delay:=PVL.Z201_Config.Target_EP101_Level.Alarm_Delay;
Burkert.Alarm_Window_Convert(window:=tAlarm,Config:=PVL.AIT[AIT_Mapping.LT_101_P].Alarm_Config);
*)


PVl.AIT[AIT_Mapping.LT_01A].Alarm_Config.Silence:=TRUE;
PVl.AIT[AIT_Mapping.LT_01B].Alarm_Config.Silence:=TRUE;
PVL.AIT[ait_Mapping.UV_001].Alarm_Config.Silence:=TRUE;

CASE PVL.Z201_Config.Task.eTask OF
	eZ201_Task.Off:
		PVl.AIT[AIT_Mapping.LT_101_P].Alarm_Config.Silence:=FALSE;
		PVl.AIT[AIT_Mapping.LT_101_T].Alarm_Config.Silence:=TRUE;
		PVL.AIT[AIT_Mapping.LT_201].Alarm_Config.Silence:=FALSE;
		PVl.AIT[AIT_Mapping.LT_201A_P].Alarm_Config.Silence:=FALSE;
		PVL.AIT[AIT_Mapping.LT_201A_T].Alarm_Config.Silence:=TRUE;
		PVL.s8312[s8312_Mapping.PT_201].Alarm_Config.Silence:=TRUE;
		PVL.s8098[s8098_Mapping.FT_201].PDO.VolumeFlow.Alarm_Config.Silence:=TRUE;
		PVL.s8098[s8098_mapping.FT_201].PDO.Temp.Alarm_Config.Silence:=TRUE;
		PVL.s8098[s8098_Mapping.FT_201].PDO.Totaliser_1.Alarm_Config.Silence:=TRUE;
		PVL.s8098[s8098_Mapping.FT_201].PDO.Totaliser_2.Alarm_Config.Silence:=TRUE;
		PVL.s8098[s8098_Mapping.FT_201].PDO.Concentration_1.Alarm_Config.Silence:=TRUE;
		PVL.s8098[s8098_Mapping.FT_201].PDO.Concentration_2.Alarm_Config.Silence:=TRUE;
		//PVL.s8050[s8050_Mapping.FT_201A].Rate_1.Alarm_Config.Silence:=TRUE;
		PVL.s8050[s8050_mapping.FT_201A].Temp.Alarm_Config.Silence:=TRUE;
		PVL.s8050[s8050_Mapping.FT_201A].CND.Alarm_Config.Silence:=TRUE;
		Burkert.Alarm_Window_Convert(window:=PVL.Z201_Config.Target_Flow,Config:=PVL.s8098[s8098_Mapping.FT_201].PDO.VolumeFlow.Alarm_Config);
	eZ201_Task.Drain:
		PVl.AIT[AIT_Mapping.LT_101_P].Alarm_Config.Silence:=FALSE;
		PVl.AIT[AIT_Mapping.LT_101_T].Alarm_Config.Silence:=TRUE;
		PVL.AIT[AIT_Mapping.LT_201].Alarm_Config.Silence:=FALSE;
		PVl.AIT[AIT_Mapping.LT_201A_P].Alarm_Config.Silence:=FALSE;
		PVL.AIT[AIT_Mapping.LT_201A_T].Alarm_Config.Silence:=TRUE;
		PVL.s8312[s8312_Mapping.PT_201].Alarm_Config.Silence:=Network.VFD[VFD_Mapping.VFD_201].Actual<VFD_Min_PCT;
		PVL.s8098[s8098_Mapping.FT_201].PDO.VolumeFlow.Alarm_Config.Silence:=Network.VFD[VFD_Mapping.VFD_201].Actual<VFD_Min_PCT;
		PVL.s8098[s8098_mapping.FT_201].PDO.Temp.Alarm_Config.Silence:=TRUE;
		PVL.s8098[s8098_Mapping.FT_201].PDO.Totaliser_1.Alarm_Config.Silence:=TRUE;
		PVL.s8098[s8098_Mapping.FT_201].PDO.Totaliser_2.Alarm_Config.Silence:=TRUE;
		PVL.s8098[s8098_Mapping.FT_201].PDO.Concentration_1.Alarm_Config.Silence:=TRUE;
		PVL.s8098[s8098_Mapping.FT_201].PDO.Concentration_2.Alarm_Config.Silence:=TRUE;
		//PVL.s8050[s8050_Mapping.FT_201A].Rate_1.Alarm_Config.Silence:=TRUE;
		PVL.s8050[s8050_mapping.FT_201A].Temp.Alarm_Config.Silence:=TRUE;
		PVL.s8050[s8050_Mapping.FT_201A].CND.Alarm_Config.Silence:=TRUE;
		Burkert.Alarm_Window_Convert(window:=PVL.Z201_Config.Drain_Rate,Config:=PVL.s8098[s8098_Mapping.FT_201].PDO.VolumeFlow.Alarm_Config);
	eZ201_Task.EP101_Level:
		PVl.AIT[AIT_Mapping.LT_101_P].Alarm_Config.Silence:=FALSE;
		PVl.AIT[AIT_Mapping.LT_101_T].Alarm_Config.Silence:=TRUE;
		PVL.AIT[AIT_Mapping.LT_201].Alarm_Config.Silence:=FALSE;
		PVl.AIT[AIT_Mapping.LT_201A_P].Alarm_Config.Silence:=FALSE;
		PVL.AIT[AIT_Mapping.LT_201A_T].Alarm_Config.Silence:=TRUE;
		PVL.s8312[s8312_Mapping.PT_201].Alarm_Config.Silence:=Network.VFD[VFD_Mapping.VFD_201].Output_Pct<VFD_Min_PCT;
		PVL.s8098[s8098_Mapping.FT_201].PDO.VolumeFlow.Alarm_Config.Silence:=TRUE;//Network.VFD[VFD_Mapping.VFD_201].Output_Pct<VFD_Min_PCT;
		PVL.s8098[s8098_mapping.FT_201].PDO.Temp.Alarm_Config.Silence:=TRUE;
		PVL.s8098[s8098_Mapping.FT_201].PDO.Totaliser_1.Alarm_Config.Silence:=TRUE;
		PVL.s8098[s8098_Mapping.FT_201].PDO.Totaliser_2.Alarm_Config.Silence:=TRUE;
		PVL.s8098[s8098_Mapping.FT_201].PDO.Concentration_1.Alarm_Config.Silence:=TRUE;
		PVL.s8098[s8098_Mapping.FT_201].PDO.Concentration_2.Alarm_Config.Silence:=TRUE;
		//PVL.s8050[s8050_Mapping.FT_201A].Rate_1.Alarm_Config.Silence:=TRUE;
		PVL.s8050[s8050_mapping.FT_201A].Temp.Alarm_Config.Silence:=TRUE;
		PVL.s8050[s8050_Mapping.FT_201A].CND.Alarm_Config.Silence:=TRUE;
		//Burkert.Alarm_Window_Convert(window:=PVL.Z201_Config.Target_Flow,Config:=PVL.s8098[s8098_Mapping.FT_201].PDO.VolumeFlow.Alarm_Config);
		Burkert.Alarm_Window_Convert(window:=PVL.Z201_Config.Drain_Rate,Config:=PVL.s8098[s8098_Mapping.FT_201].PDO.VolumeFlow.Alarm_Config);
	eZ201_Task.Flow:
		PVl.AIT[AIT_Mapping.LT_101_P].Alarm_Config.Silence:=FALSE;
		PVl.AIT[AIT_Mapping.LT_101_T].Alarm_Config.Silence:=TRUE;
		PVL.AIT[AIT_Mapping.LT_201].Alarm_Config.Silence:=FALSE;
		PVl.AIT[AIT_Mapping.LT_201A_P].Alarm_Config.Silence:=FALSE;
		PVL.AIT[AIT_Mapping.LT_201A_T].Alarm_Config.Silence:=TRUE;
		PVL.s8312[s8312_Mapping.PT_201].Alarm_Config.Silence:=Network.VFD[VFD_Mapping.VFD_201].Output_Pct<VFD_Min_PCT;
		PVL.s8098[s8098_Mapping.FT_201].PDO.VolumeFlow.Alarm_Config.Silence:=Network.VFD[VFD_Mapping.VFD_201].Output_Pct<VFD_Min_PCT;
		PVL.s8098[s8098_mapping.FT_201].PDO.Temp.Alarm_Config.Silence:=TRUE;
		PVL.s8098[s8098_Mapping.FT_201].PDO.Totaliser_1.Alarm_Config.Silence:=TRUE;
		PVL.s8098[s8098_Mapping.FT_201].PDO.Totaliser_2.Alarm_Config.Silence:=TRUE;
		PVL.s8098[s8098_Mapping.FT_201].PDO.Concentration_1.Alarm_Config.Silence:=TRUE;
		PVL.s8098[s8098_Mapping.FT_201].PDO.Concentration_2.Alarm_Config.Silence:=TRUE;
		//PVL.s8050[s8050_Mapping.FT_201A].Rate_1.Alarm_Config.Silence:=TRUE;
		PVL.s8050[s8050_mapping.FT_201A].Temp.Alarm_Config.Silence:=TRUE;
		PVL.s8050[s8050_Mapping.FT_201A].CND.Alarm_Config.Silence:=TRUE;
		Burkert.Alarm_Window_Convert(window:=PVL.Z201_Config.Target_Flow,Config:=PVL.s8098[s8098_Mapping.FT_201].PDO.VolumeFlow.Alarm_Config);
	eZ201_Task.TK201_Level:
		PVl.AIT[AIT_Mapping.LT_101_P].Alarm_Config.Silence:=FALSE;
		PVl.AIT[AIT_Mapping.LT_101_T].Alarm_Config.Silence:=TRUE;
		PVL.AIT[AIT_Mapping.LT_201].Alarm_Config.Silence:=FALSE;
		PVl.AIT[AIT_Mapping.LT_201A_P].Alarm_Config.Silence:=FALSE;
		PVL.AIT[AIT_Mapping.LT_201A_T].Alarm_Config.Silence:=TRUE;
		PVL.s8312[s8312_Mapping.PT_201].Alarm_Config.Silence:=Network.VFD[VFD_Mapping.VFD_201].Output_Pct<VFD_Min_PCT;
		PVL.s8098[s8098_Mapping.FT_201].PDO.VolumeFlow.Alarm_Config.Silence:=TRUE;//Network.VFD[VFD_Mapping.VFD_201].Output_Pct<VFD_Min_PCT;
		PVL.s8098[s8098_mapping.FT_201].PDO.Temp.Alarm_Config.Silence:=TRUE;
		PVL.s8098[s8098_Mapping.FT_201].PDO.Totaliser_1.Alarm_Config.Silence:=TRUE;
		PVL.s8098[s8098_Mapping.FT_201].PDO.Totaliser_2.Alarm_Config.Silence:=TRUE;
		PVL.s8098[s8098_Mapping.FT_201].PDO.Concentration_1.Alarm_Config.Silence:=TRUE;
		PVL.s8098[s8098_Mapping.FT_201].PDO.Concentration_2.Alarm_Config.Silence:=TRUE;
		//PVL.s8050[s8050_Mapping.FT_201A].Rate_1.Alarm_Config.Silence:=TRUE;
		PVL.s8050[s8050_mapping.FT_201A].Temp.Alarm_Config.Silence:=TRUE;
		PVL.s8050[s8050_Mapping.FT_201A].CND.Alarm_Config.Silence:=TRUE;
		Burkert.Alarm_Window_Convert(window:=PVL.Z201_Config.Target_Flow,Config:=PVL.s8098[s8098_Mapping.FT_201].PDO.VolumeFlow.Alarm_Config);
	eZ201_Task.Z100_Flow:
		PVl.AIT[AIT_Mapping.LT_101_P].Alarm_Config.Silence:=FALSE;
		PVl.AIT[AIT_Mapping.LT_101_T].Alarm_Config.Silence:=TRUE;
		PVL.AIT[AIT_Mapping.LT_201].Alarm_Config.Silence:=FALSE;
		PVl.AIT[AIT_Mapping.LT_201A_P].Alarm_Config.Silence:=FALSE;
		PVL.AIT[AIT_Mapping.LT_201A_T].Alarm_Config.Silence:=TRUE;
		PVL.s8312[s8312_Mapping.PT_201].Alarm_Config.Silence:=Network.VFD[VFD_Mapping.VFD_201].Output_Pct<VFD_Min_PCT;
		PVL.s8098[s8098_Mapping.FT_201].PDO.VolumeFlow.Alarm_Config.Silence:=Network.VFD[VFD_Mapping.VFD_201].Output_Pct<VFD_Min_PCT;
		PVL.s8098[s8098_mapping.FT_201].PDO.Temp.Alarm_Config.Silence:=TRUE;
		PVL.s8098[s8098_Mapping.FT_201].PDO.Totaliser_1.Alarm_Config.Silence:=TRUE;
		PVL.s8098[s8098_Mapping.FT_201].PDO.Totaliser_2.Alarm_Config.Silence:=TRUE;
		PVL.s8098[s8098_Mapping.FT_201].PDO.Concentration_1.Alarm_Config.Silence:=TRUE;
		PVL.s8098[s8098_Mapping.FT_201].PDO.Concentration_2.Alarm_Config.Silence:=TRUE;
		//PVL.s8050[s8050_Mapping.FT_201A].Rate_1.Alarm_Config.Silence:=TRUE;
		PVL.s8050[s8050_mapping.FT_201A].Temp.Alarm_Config.Silence:=TRUE;
		PVL.s8050[s8050_Mapping.FT_201A].CND.Alarm_Config.Silence:=TRUE;
		PVL.s8098[s8098_Mapping.FT_201].PDO.VolumeFlow.Alarm_Config:=PVL.s8098[s8098_Mapping.FT_101].PDO.VolumeFlow.Alarm_Config;
	eZ201_Task.Z202_Flow:
		PVl.AIT[AIT_Mapping.LT_101_P].Alarm_Config.Silence:=FALSE;
		PVl.AIT[AIT_Mapping.LT_101_T].Alarm_Config.Silence:=TRUE;
		PVL.AIT[AIT_Mapping.LT_201].Alarm_Config.Silence:=FALSE;
		PVl.AIT[AIT_Mapping.LT_201A_P].Alarm_Config.Silence:=FALSE;
		PVL.AIT[AIT_Mapping.LT_201A_T].Alarm_Config.Silence:=TRUE;
		PVL.s8312[s8312_Mapping.PT_201].Alarm_Config.Silence:=Network.VFD[VFD_Mapping.VFD_201].Output_Pct<VFD_Min_PCT;
		PVL.s8098[s8098_Mapping.FT_201].PDO.VolumeFlow.Alarm_Config.Silence:=Network.VFD[VFD_Mapping.VFD_201].Output_Pct<VFD_Min_PCT;
		PVL.s8098[s8098_mapping.FT_201].PDO.Temp.Alarm_Config.Silence:=TRUE;
		PVL.s8098[s8098_Mapping.FT_201].PDO.Totaliser_1.Alarm_Config.Silence:=TRUE;
		PVL.s8098[s8098_Mapping.FT_201].PDO.Totaliser_2.Alarm_Config.Silence:=TRUE;
		PVL.s8098[s8098_Mapping.FT_201].PDO.Concentration_1.Alarm_Config.Silence:=TRUE;
		PVL.s8098[s8098_Mapping.FT_201].PDO.Concentration_2.Alarm_Config.Silence:=TRUE;
		//PVL.s8050[s8050_Mapping.FT_201A].Rate_1.Alarm_Config.Silence:=TRUE;
		PVL.s8050[s8050_mapping.FT_201A].Temp.Alarm_Config.Silence:=TRUE;
		PVL.s8050[s8050_Mapping.FT_201A].CND.Alarm_Config.Silence:=TRUE;
		PVL.s8098[s8098_mapping.FT_201].PDO.VolumeFlow.Alarm_Config:=PVL.s8098[s8098_Mapping.FT_203].PDO.VolumeFlow.Alarm_Config;
eZ201_Task.Agitate_only:
		PVl.AIT[AIT_Mapping.LT_101_P].Alarm_Config.Silence:=FALSE;
		PVl.AIT[AIT_Mapping.LT_101_T].Alarm_Config.Silence:=TRUE;
		PVL.AIT[AIT_Mapping.LT_201].Alarm_Config.Silence:=FALSE;
		PVl.AIT[AIT_Mapping.LT_201A_P].Alarm_Config.Silence:=FALSE;
		PVL.AIT[AIT_Mapping.LT_201A_T].Alarm_Config.Silence:=TRUE;
		PVL.s8312[s8312_Mapping.PT_201].Alarm_Config.Silence:=Network.VFD[VFD_Mapping.VFD_201].Output_Pct<VFD_Min_PCT;
		PVL.s8098[s8098_Mapping.FT_201].PDO.VolumeFlow.Alarm_Config.Silence:=True;//Network.VFD[VFD_Mapping.VFD_201].Output_Pct<VFD_Min_PCT;
		PVL.s8098[s8098_mapping.FT_201].PDO.Temp.Alarm_Config.Silence:=TRUE;
		PVL.s8098[s8098_Mapping.FT_201].PDO.Totaliser_1.Alarm_Config.Silence:=TRUE;
		PVL.s8098[s8098_Mapping.FT_201].PDO.Totaliser_2.Alarm_Config.Silence:=TRUE;
		PVL.s8098[s8098_Mapping.FT_201].PDO.Concentration_1.Alarm_Config.Silence:=TRUE;
		PVL.s8098[s8098_Mapping.FT_201].PDO.Concentration_2.Alarm_Config.Silence:=TRUE;
		//PVL.s8050[s8050_Mapping.FT_201A].Rate_1.Alarm_Config.Silence:=TRUE;
		PVL.s8050[s8050_mapping.FT_201A].Temp.Alarm_Config.Silence:=TRUE;
		PVL.s8050[s8050_Mapping.FT_201A].CND.Alarm_Config.Silence:=TRUE;
		Burkert.Alarm_Window_Convert(window:=PVL.Z201_Config.Drain_Rate,Config:=PVL.s8098[s8098_Mapping.FT_201].PDO.VolumeFlow.Alarm_Config);

		
END_CASE



PVL.Z201_Config.Mixer_Motor_Current.Debounce:=1;
PVL.Z201_Config.Mixer_Motor_Current.Hi_Warn:=PVL.Z201_Config.Mixer_Motor_Current.Hi_Hi_Alarm-0.001;
PVL.Z201_Config.Mixer_Motor_Current.Hi_Norm :=PVL.Z201_Config.Mixer_Motor_Current.Hi_Hi_Alarm-0.002;
PVL.Z201_Config.Mixer_Motor_Current.Low_Norm:=(-1);
PVL.Z201_Config.Mixer_Motor_Current.Low_warn:=(-2);
PVL.Z201_Config.Mixer_Motor_Current.Low_Low_Alarm:=(-3);

PVl.s8050[s8050_mapping.FT_201A].Rate_1.Alarm_Config.Silence:=PVL.s8098[s8098_Mapping.FT_201].PDO.VolumeFlow.Alarm_Config.Silence;
PVL.Z201_Config.READY:=(Local_Status=PVl.Z201_Config.Status.eStatus);

	


              
END_ACTION

ACTION Evaluate_Task_Flow:
                tStatus:=Local_Status;

IF GVl.LS[LS_Mapping.LSLL_202].Status.eStatus=Burkert.DI_Status.No_Liquid_Detected_Alarm THEN tStatus:=eZ201_Status.Pump_Intake_Dry_LSLL202; END_IF;
IF GVl.LS[LS_Mapping.LSHH_204 ].Status.eStatus=Burkert.DI_Status.Liquid_Detected_Alarm THEN tStatus:=eZ201_Status.TK201_LSHH204_High_High_Level_Alarm; END_IF;

//IF NOT(Network.VFD[VFD_Mapping.VFD_102A].Ready) THEN tStatus:=eZ201_Status.VFD_102A_Not_Ready;	END_IF;
//IF NOT(Network.VFD[VFD_Mapping.VFD_102B].Ready) THEN tStatus:=eZ201_Status.VFD_102B_Not_Ready;	END_IF;
//IF NOT(Network.VFD[VFD_Mapping.VFD_102C].Ready) THEN tStatus:=eZ201_Status.VFD_102C_Not_Ready;	END_IF;
//IF NOT(Network.VFD[VFD_Mapping.VFD_102D].Ready) THEN tStatus:=eZ201_Status.VFD_102D_Not_Ready;	END_IF;
//IF NOT(Network.VFD[VFD_Mapping.VFD_102E].Ready) THEN tStatus:=eZ201_Status.VFD_102E_Not_Ready;	END_IF;
//IF NOT(Network.VFD[VFD_Mapping.VFD_102F].Ready) THEN tStatus:=eZ201_Status.VFD_102F_Not_Ready;	END_IF;
//IF NOT(Network.VFD[VFD_Mapping.VFD_102G].Ready) THEN tStatus:=eZ201_Status.VFD_102G_Not_Ready;	END_IF;
//IF NOT(Network.VFD[VFD_Mapping.VFD_102H].Ready) THEN tStatus:=eZ201_Status.VFD_102H_Not_Ready;	END_IF;
IF NOT(Network.VFD[VFD_Mapping.VFD_201].Ready) THEN tStatus:=eZ201_Status.VFD_201_Not_Ready;	END_IF;
//IF Network.VFD[VFD_Mapping.VFD_102A].Status=Burkert.eVFD_Status.High_High_Current_Alarm THEN tStatus:=eZ201_Status.VFD_102A_High_Current;	END_IF;
//IF Network.VFD[VFD_Mapping.VFD_102B].Status=Burkert.eVFD_Status.High_High_Current_Alarm THEN tStatus:=eZ201_Status.VFD_102B_High_Current;	END_IF;/
//IF Network.VFD[VFD_Mapping.VFD_102C].Status=Burkert.eVFD_Status.High_High_Current_Alarm THEN tStatus:=eZ201_Status.VFD_102C_High_Current;	END_IF;
//IF Network.VFD[VFD_Mapping.VFD_102D].Status=Burkert.eVFD_Status.High_High_Current_Alarm THEN tStatus:=eZ201_Status.VFD_102D_High_Current;	END_IF;
//IF Network.VFD[VFD_Mapping.VFD_102E].Status=Burkert.eVFD_Status.High_High_Current_Alarm THEN tStatus:=eZ201_Status.VFD_102E_High_Current;	END_IF;
//IF Network.VFD[VFD_Mapping.VFD_102F].Status=Burkert.eVFD_Status.High_High_Current_Alarm THEN tStatus:=eZ201_Status.VFD_102F_High_Current;	END_IF;
//IF Network.VFD[VFD_Mapping.VFD_102G].Status=Burkert.eVFD_Status.High_High_Current_Alarm THEN tStatus:=eZ201_Status.VFD_102G_High_Current;	END_IF;
//IF Network.VFD[VFD_Mapping.VFD_102H].Status=Burkert.eVFD_Status.High_High_Current_Alarm THEN tStatus:=eZ201_Status.VFD_102H_High_Current;	END_IF;


IF NOT(GVL.s3363[s3363_mapping.ACV_201].Ready) THEN	tStatus:=eZ201_Status.ACV_201_Not_Ready;	END_IF;
	
IF NOT(PVl.s8312[s8312_mapping.PT_201].Ready) THEN	tStatus:=eZ201_status.PT201_Not_Ready;	END_IF;
IF PVL.s8312[s8312_Mapping.PT_201].Status.eStatus=Burkert.eSensor_Status.HiHi_Alarm THEN tStatus:=eZ201_Status.PT201_High_Pressure_Alarm; END_IF;
//IF PVL.s8312[s8312_Mapping.PT_201].Status.eStatus=Burkert.eSensor_Status.Low_Low_Alarm THEN tStatus:=eZ201_Status.PT201_Low_Pressure_Alarm; END_IF;

IF NOT(PVL.s8098[s8098_Mapping.FT_201].Ready) THEN	tStatus:=eZ201_status.FT201_Not_Ready;	END_IF;
IF PVL.s8098[s8098_Mapping.FT_201].PDO.VolumeFlow.Status.eStatus=Burkert.eSensor_Status.Low_Low_Alarm THEN tStatus:=eZ201_status.FT201_Low_Low_Flow_Alarm;	END_IF;

//IF NOT(PVL.AIT[AIT_Mapping.LT_101_P].Ready) THEN tStatus:=eZ201_Status.LT101_Not_Ready;	END_IF;
//IF NOT(PVL.AIT[AIT_Mapping.LT_201A_P].Ready) THEN tStatus:=eZ201_Status.LT201A_Not_Ready;	END_IF;
IF NOT(PVL.AIT[AIT_Mapping.LT_201].Ready) THEN tStatus:=eZ201_Status.LT201_Not_Ready;	END_IF;
IF NOT(PVL.AIT[AIT_Mapping.LT_202].Ready) THEN tStatus:=eZ201_Status.LT202_Not_Ready;	END_IF;
//IF NOT(PVL.AIT[AIT_Mapping.LT_202a].Ready) THEN tStatus:=eZ201_Status.LT202a_Not_Ready;	END_IF;

//IF PVL.AIT[AIT_Mapping.LT_101_P].Status.eStatus=Burkert.eSensor_Status.HiHi_Alarm THEN	tStatus:=eZ201_Status.LT101_High_High_Alarm; END_IF;
///IF PVL.AIT[AIT_Mapping.LT_101_P].Status.eStatus=Burkert.eSensor_Status.Low_Low_Alarm THEN	tStatus:=eZ201_Status.LT101_Low_Low_Alarm; END_IF;

//IF PVL.AIT[AIT_Mapping.LT_201A_P].Status.eStatus=Burkert.eSensor_Status.HiHi_Alarm THEN	tStatus:=eZ201_Status.LT201A_High_High_Alarm; END_IF;
//IF PVL.AIT[AIT_Mapping.LT_201A_P].Status.eStatus=Burkert.eSensor_Status.Low_Low_Alarm THEN	tStatus:=eZ201_Status.LT201A_Low_Low_Alarm; END_IF;

//IF PVL.AIT[AIT_Mapping.LT_201].Status.eStatus=Burkert.eSensor_Status.HiHi_Alarm THEN	tStatus:=eZ201_Status.LT201_High_High_Alarm; END_IF;
IF PVL.AIT[AIT_Mapping.LT_201].Status.eStatus=Burkert.eSensor_Status.Low_Low_Alarm THEN	tStatus:=eZ201_Status.LT201_Low_Low_Alarm; END_IF;
//IF PVL.AIT[AIT_Mapping.LT_202].Status.eStatus=Burkert.eSensor_Status.HiHi_Alarm THEN	tStatus:=eZ201_Status.LT202_High_High_Alarm; END_IF;
IF PVL.AIT[AIT_Mapping.LT_202a].Status.eStatus=Burkert.eSensor_Status.HiHi_Alarm THEN	tStatus:=eZ201_Status.LT202a_High_High_Alarm; END_IF;

IF PVl.s8312[s8312_mapping.PT_201].Status.eStatus=Burkert.eSensor_Status.Low_Low_Alarm 					THEN	tStatus:=eZ201_Status.PT201_Low_Pressure_Alarm; END_IF;
IF PVl.s8312[s8312_mapping.PT_201].Status.eStatus=Burkert.eSensor_Status.HiHi_Alarm 					THEN	tStatus:=eZ201_Status.PT201_High_Pressure_Alarm; END_IF;
IF PVL.s8098[s8098_Mapping.FT_201].PDO.VolumeFlow.Status.eStatus=Burkert.eSensor_Status.Low_Low_Alarm	THEN	tStatus:=ez201_Status.FT201_Low_Low_Flow_Alarm; END_IF;

PVL.Z201_Config.Status.eStatus:=tStatus;

              
END_ACTION

ACTION Evaluate_Agitate:
                tStatus:=Local_Status;

//IF GVl.LS[LS_Mapping.LSLL_202].Status.eStatus=Burkert.DI_Status.No_Liquid_Detected_Alarm THEN tStatus:=eZ201_Status.Pump_Intake_Dry_LSLL202; END_IF;
//IF GVl.LS[LS_Mapping.LSHH_204 ].Status.eStatus=Burkert.DI_Status.Liquid_Detected_Alarm THEN tStatus:=eZ201_Status.TK201_LSHH204_High_High_Level_Alarm; END_IF;

//IF NOT(Network.VFD[VFD_Mapping.VFD_102A].Ready) THEN tStatus:=eZ201_Status.VFD_102A_Not_Ready;	END_IF;
//IF NOT(Network.VFD[VFD_Mapping.VFD_102B].Ready) THEN tStatus:=eZ201_Status.VFD_102B_Not_Ready;	END_IF;
// NOT(Network.VFD[VFD_Mapping.VFD_102C].Ready) THEN tStatus:=eZ201_Status.VFD_102C_Not_Ready;	END_IF;
//IF NOT(Network.VFD[VFD_Mapping.VFD_102D].Ready) THEN tStatus:=eZ201_Status.VFD_102D_Not_Ready;	END_IF;
//IF NOT(Network.VFD[VFD_Mapping.VFD_102E].Ready) THEN tStatus:=eZ201_Status.VFD_102E_Not_Ready;	END_IF;
//IF NOT(Network.VFD[VFD_Mapping.VFD_102F].Ready) THEN tStatus:=eZ201_Status.VFD_102F_Not_Ready;	END_IF;
//IF NOT(Network.VFD[VFD_Mapping.VFD_102G].Ready) THEN tStatus:=eZ201_Status.VFD_102G_Not_Ready;	END_IF;
//IF NOT(Network.VFD[VFD_Mapping.VFD_102H].Ready) THEN tStatus:=eZ201_Status.VFD_102H_Not_Ready;	END_IF;

IF Network.VFD[VFD_Mapping.VFD_102A].Status=Burkert.eVFD_Status.High_High_Current_Alarm THEN tStatus:=eZ201_Status.VFD_102A_High_Current;	END_IF;
IF Network.VFD[VFD_Mapping.VFD_102B].Status=Burkert.eVFD_Status.High_High_Current_Alarm THEN tStatus:=eZ201_Status.VFD_102B_High_Current;	END_IF;
IF Network.VFD[VFD_Mapping.VFD_102C].Status=Burkert.eVFD_Status.High_High_Current_Alarm THEN tStatus:=eZ201_Status.VFD_102C_High_Current;	END_IF;
IF Network.VFD[VFD_Mapping.VFD_102D].Status=Burkert.eVFD_Status.High_High_Current_Alarm THEN tStatus:=eZ201_Status.VFD_102D_High_Current;	END_IF;
//IF Network.VFD[VFD_Mapping.VFD_102E].Status=Burkert.eVFD_Status.High_High_Current_Alarm THEN tStatus:=eZ201_Status.VFD_102E_High_Current;	END_IF;
//IF Network.VFD[VFD_Mapping.VFD_102F].Status=Burkert.eVFD_Status.High_High_Current_Alarm THEN tStatus:=eZ201_Status.VFD_102F_High_Current;	END_IF;
//IF Network.VFD[VFD_Mapping.VFD_102G].Status=Burkert.eVFD_Status.High_High_Current_Alarm THEN tStatus:=eZ201_Status.VFD_102G_High_Current;	END_IF;
//IF Network.VFD[VFD_Mapping.VFD_102H].Status=Burkert.eVFD_Status.High_High_Current_Alarm THEN tStatus:=eZ201_Status.VFD_102H_High_Current;	END_IF;


//IF NOT(Network.VFD[VFD_Mapping.VFD_201].Ready) THEN tStatus:=eZ201_Status.VFD_201_Not_Ready;	END_IF;

//IF NOT(GVL.s3363[s3363_mapping.ACV_201].Ready) THEN	tStatus:=eZ201_Status.ACV_201_Not_Ready;	END_IF;
	
///IF NOT(PVl.s8312[s8312_mapping.PT_201].Ready) THEN	tStatus:=eZ201_status.PT201_Not_Ready;	END_IF;
//IF NOT(PVL.s8098[s8098_Mapping.FT_201].Ready) THEN	tStatus:=eZ201_status.FT201_Not_Ready;	END_IF;


IF NOT(PVL.AIT[AIT_Mapping.LT_101_P].Ready) THEN tStatus:=eZ201_Status.LT101_Not_Ready;	END_IF;
//IF NOT(PVL.AIT[AIT_Mapping.LT_201A_P].Ready) THEN tStatus:=eZ201_Status.LT201A_Not_Ready;	END_IF;
//IF NOT(PVL.AIT[AIT_Mapping.LT_201].Ready) THEN tStatus:=eZ201_Status.LT201_Not_Ready;	END_IF;

///IF PVL.AIT[AIT_Mapping.LT_101_P].Status.eStatus=Burkert.eSensor_Status.HiHi_Alarm THEN	tStatus:=eZ201_Status.LT101_High_High_Alarm; END_IF;
IF PVL.AIT[AIT_Mapping.LT_101_P].Status.eStatus=Burkert.eSensor_Status.Low_Low_Alarm THEN	tStatus:=eZ201_Status.LT101_Low_Low_Alarm; END_IF;

//IF PVL.AIT[AIT_Mapping.LT_201A_P].Status.eStatus=Burkert.eSensor_Status.HiHi_Alarm THEN	tStatus:=eZ201_Status.LT201A_High_High_Alarm; END_IF;
//IF PVL.AIT[AIT_Mapping.LT_201A_P].Status.eStatus=Burkert.eSensor_Status.Low_Low_Alarm THEN	tStatus:=eZ201_Status.LT201A_Low_Low_Alarm; END_IF;

//IF PVL.AIT[AIT_Mapping.LT_201].Status.eStatus=Burkert.eSensor_Status.HiHi_Alarm THEN	tStatus:=eZ201_Status.LT201_High_High_Alarm; END_IF;
//IF PVL.AIT[AIT_Mapping.LT_201].Status.eStatus=Burkert.eSensor_Status.Low_Low_Alarm THEN	tStatus:=eZ201_Status.LT201_Low_Low_Alarm; END_IF;


PVL.Z201_Config.Status.eStatus:=tStatus;

              
END_ACTION

ACTION Task_agitate:
                IF PVL.Z201_Config.Task.eTask<> Local_Task THEN
	Local_Task:=PVL.Z201_Config.Task.eTask;
	Local_Status:=eZ201_Status.Agitate_Only;
END_IF;


CASE PVL.Z201_Config.Status.eStatus OF
	//eZ201_Status.LT101_High_High_Alarm:			Local_Status:=PVL.Z201_Config.Status.eStatus;
	//eZ201_Status.LT101_Low_Low_Alarm:			Local_Status:=PVL.Z201_Config.Status.eStatus;
	//eZ201_Status.LT201_High_High_Alarm:			Local_Status:=PVL.Z201_Config.Status.eStatus;
	//eZ201_Status.LT201_Low_Low_Alarm:			Local_Status:=PVL.Z201_Config.Status.eStatus;
	//eZ201_Status.LT201A_High_High_Alarm:		Local_Status:=PVL.Z201_Config.Status.eStatus;
	//eZ201_Status.LT201A_Low_Low_Alarm:			Local_Status:=PVL.Z201_Config.Status.eStatus;
	//eZ201_Status.TK201_LSHH204_High_High_Level_Alarm:	Local_Status:=PVL.Z201_Config.Status.eStatus;
	//eZ201_Status.Pump_Intake_Dry_LSLL202:		Local_Status:=PVL.Z201_Config.Status.eStatus;
	//eZ201_Status.PT201_High_Pressure_Alarm:		Local_Status:=PVL.Z201_Config.Status.eStatus;
	///eZ201_Status.PT201_Low_Pressure_Alarm:		Local_Status:=PVL.Z201_Config.Status.eStatus;
	//eZ201_Status.FT201_Low_Low_Flow_Alarm:		Local_Status:=PVL.Z201_Config.Status.eStatus;
	
	eZ201_Status.LT201_Low_Low_Alarm:		IF Level_ton.Q THEN local_Status:= eZ201_Status.Waiting_For_Level_OK_LT201; END_IF;
	eZ201_Status.LT202_High_High_Alarm:		IF Level_ton.Q THEN local_Status:= eZ201_Status.Waiting_For_Level_OK_LT202; END_IF;
	eZ201_Status.Waiting_For_Level_OK_LT201:	IF PVL.AIT[AIT_Mapping.LT_201].Status.eStatus=Burkert.eSensor_Status.OK THEN Local_Task:=999; END_IF;
	eZ201_Status.Waiting_For_Level_OK_LT202:	IF PVL.AIT[AIT_Mapping.LT_202].Status.eStatus=Burkert.eSensor_Status.OK THEN Local_Task:=999; END_IF;
	
	
	eZ201_Status.PT201_High_Pressure_Alarm:		Local_Status:=PVL.Z201_Config.Status.eStatus;
	eZ201_Status.PT201_Low_Pressure_Alarm:		Local_Status:=PVL.Z201_Config.Status.eStatus;
	eZ201_Status.FT201_Low_Low_Flow_Alarm:		Local_Status:=PVL.Z201_Config.Status.eStatus;
	

END_CASE;

Evaluate_Agitate();
              
END_ACTION
END_PROGRAM

PROGRAM PID_Manager
  VAR
    Z100_Flow_CTRL : Burkert.PID_UDFB;
    Z100_Level_CTRL : Burkert.PID_UDFB;
    Z100_Pressure_CTRL : Burkert.PID_UDFB;
    Z201_EP101_Level_ctrl : Burkert.PID_UDFB;
    Z201_Flow_ctrl : Burkert.PID_UDFB;
    Z201_TK201_Level_ctrl : Burkert.PID_UDFB;
    Z202_EP101_Level_ctrl : Burkert.PID_UDFB;
    Z202_TK201_Level_ctrl : Burkert.PID_UDFB;
    Z202_Flow_ctrl : Burkert.PID_UDFB;
    Z202_Recovery_Level_ctrl : Burkert.PID_UDFB;
    Z202_Filter_Flow_ctrl : Burkert.PID_UDFB;
  END_VAR

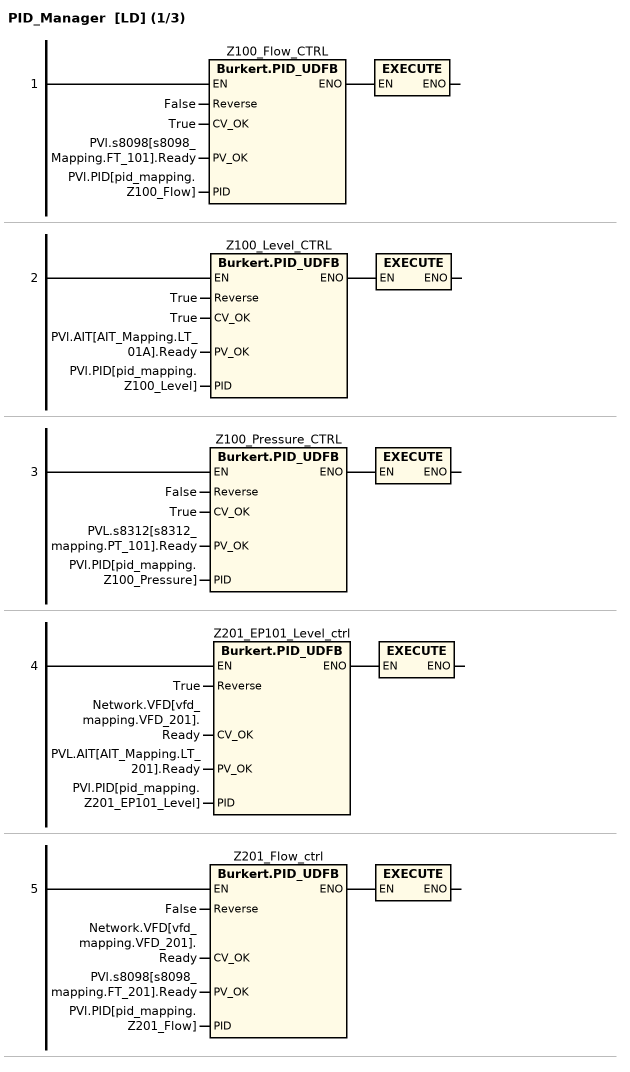
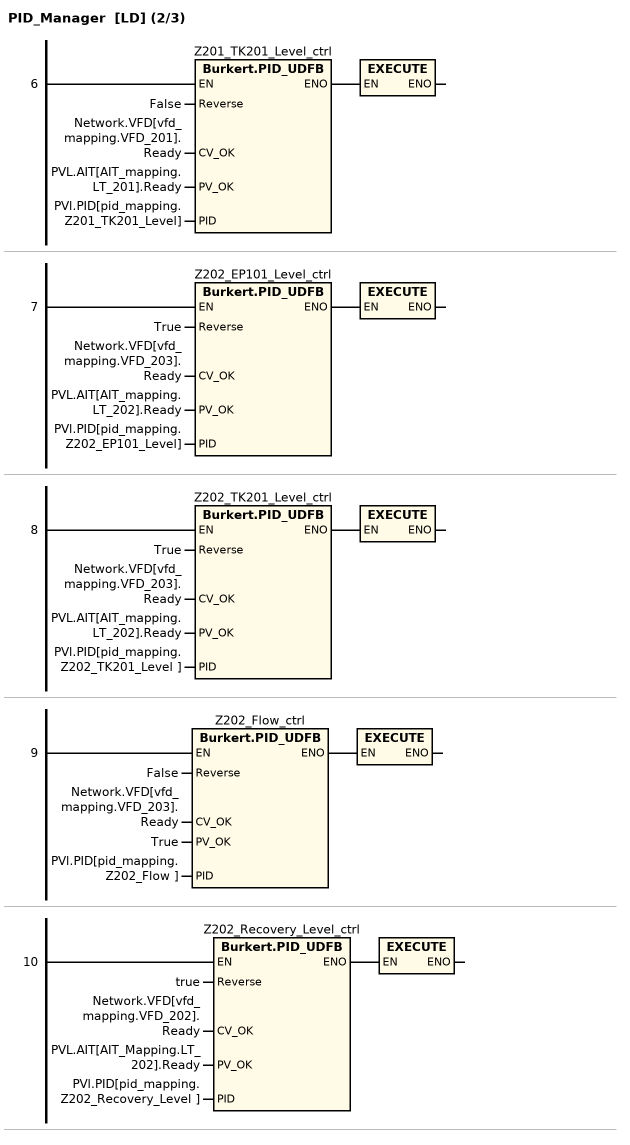
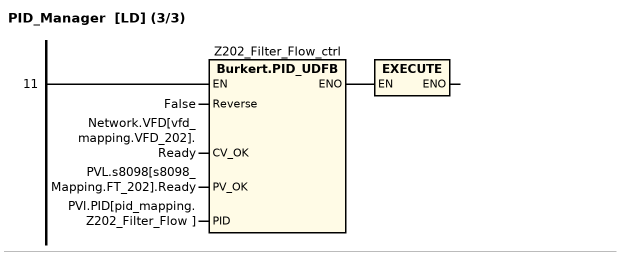
(* LD diagram, written out as Structured Text *)

Z100_Flow_CTRL(Reverse := False, CV_OK := True, PV_OK := PVl.s8098[s8098_Mapping.FT_101].Ready, PID := PVl.PID[pid_mapping.Z100_Flow]);
IF Z100_Flow_CTRL.ENO THEN
  PVl.PID[pid_mapping.Z100_Flow].InHibit:=(
  	GVL.LS[LS_Mapping.LSHH_201].Status.eStatus=Burkert.DI_Status.Liquid_Detected_Alarm
  	);
  	
  //PVl.PID[pid_mapping.Z100_Flow].Actual:=PVl.s8098[s8098_mapping.FT_101].PDO.VolumeFlow.EU;
END_IF;

Z100_Level_CTRL(Reverse := True, CV_OK := True, PV_OK := PVl.AIT[AIT_Mapping.LT_01A].Ready, PID := PVl.PID[pid_mapping.Z100_Level]);
IF Z100_Level_CTRL.ENO THEN
  PVl.PID[pid_mapping.Z100_Level].InHibit:=(
  	GVL.LS[LS_Mapping.LSHH_201].Status.eStatus=Burkert.DI_Status.Liquid_Detected_Alarm
  	);
  	
  PVl.PID[pid_mapping.Z100_Level].Actual:=PVL.AIT[AIT_Mapping.LT_01A].PCT_Scale;
END_IF;

Z100_Pressure_CTRL(Reverse := False, CV_OK := True, PV_OK := PVL.s8312[s8312_mapping.PT_101].Ready, PID := PVl.PID[pid_mapping.Z100_Pressure]);
IF Z100_Pressure_CTRL.ENO THEN
  PVl.PID[pid_mapping.Z100_Pressure].InHibit:=(
  	GVL.LS[LS_Mapping.LSHH_201].Status.eStatus=Burkert.DI_Status.Liquid_Detected_Alarm
  	);
  	
  
  PVl.PID[pid_mapping.Z100_Pressure].Actual:=PVL.s8312[s8312_mapping.PT_101].EU;
END_IF;


Z201_EP101_Level_ctrl(Reverse := True, CV_OK := Network.VFD[vfd_mapping.VFD_201].Ready, PV_OK := PVL.AIT[AIT_Mapping.LT_201].Ready, PID := PVl.PID[pid_mapping.Z201_EP101_Level]);
IF Z201_EP101_Level_ctrl.ENO THEN
  PVl.PID[pid_mapping.Z201_EP101_Level].InHibit:=(
  	GVL.LS[LS_Mapping.LSHH_204].Status.eStatus=Burkert.DI_Status.Liquid_Detected_Alarm
  	);
  	
  
  PVl.PID[pid_mapping.Z201_EP101_Level].Actual:=PVL.ait[AIT_Mapping.LT_201].PCT_Scale;
END_IF;

Z201_Flow_ctrl(Reverse := False, CV_OK := Network.VFD[vfd_mapping.VFD_201].Ready, PV_OK := PVl.s8098[s8098_mapping.FT_201].Ready, PID := PVl.PID[pid_mapping.Z201_Flow]);
IF Z201_Flow_ctrl.ENO THEN
  PVl.PID[pid_mapping.Z201_Flow].InHibit:=(
  	GVL.LS[LS_Mapping.LSHH_204].Status.eStatus=Burkert.DI_Status.Liquid_Detected_Alarm
  	);
  	
  
  //PVl.PID[pid_mapping.Z201_Flow].Actual:=PVl.s8098[s8098_mapping.FT_201].PDO.VolumeFlow.EU;
END_IF;

Z201_TK201_Level_ctrl(Reverse := False, CV_OK := Network.VFD[vfd_mapping.VFD_201].Ready, PV_OK := PVL.AIT[AIT_mapping.LT_201].Ready, PID := PVl.PID[pid_mapping.Z201_TK201_Level]);
IF Z201_TK201_Level_ctrl.ENO THEN
  PVl.PID[pid_mapping.Z201_TK201_Level].InHibit:=(
  	GVL.LS[LS_Mapping.LSHH_204].Status.eStatus=Burkert.DI_Status.Liquid_Detected_Alarm
  	);
  	
  
  PVl.PID[pid_mapping.Z201_TK201_Level].Actual:=PVL.AIT[AIT_mapping.LT_202].PCT_Scale;
END_IF;

Z202_EP101_Level_ctrl(Reverse := True, CV_OK := Network.VFD[vfd_mapping.VFD_203].Ready, PV_OK := PVL.AIT[AIT_mapping.LT_202].Ready, PID := PVl.PID[pid_mapping.Z202_EP101_Level]);
IF Z202_EP101_Level_ctrl.ENO THEN
  PVl.PID[pid_mapping.Z202_Ep101_Level].InHibit:=(
  	GVL.LS[LS_Mapping.LSHH_204].Status.eStatus=Burkert.DI_Status.Liquid_Detected_Alarm
  	);
  	
  
  PVl.PID[pid_mapping.Z202_EP101_Level].Actual:=PVL.AIT[AIT_mapping.LT_101_P].PCT_Scale;
END_IF;

Z202_TK201_Level_ctrl(Reverse := True, CV_OK := Network.VFD[vfd_mapping.VFD_203].Ready, PV_OK := PVL.AIT[AIT_mapping.LT_202].Ready, PID := PVl.PID[pid_mapping.Z202_TK201_Level ]);
IF Z202_TK201_Level_ctrl.ENO THEN
  PVl.PID[pid_mapping.Z202_TK201_Level].InHibit:=(
  	GVL.LS[LS_Mapping.LSHH_204].Status.eStatus=Burkert.DI_Status.Liquid_Detected_Alarm
  	);
  	
  
  PVl.PID[pid_mapping.Z202_Tk201_Level].Actual:=PVL.AIT[AIT_mapping.LT_202].PCT_Scale;
END_IF;

Z202_Flow_ctrl(Reverse := False, CV_OK := Network.VFD[vfd_mapping.VFD_203].Ready, PV_OK := True, PID := PVl.PID[pid_mapping.Z202_Flow ]);
IF Z202_Flow_ctrl.ENO THEN
  PVl.PID[pid_mapping.Z202_Flow].InHibit:=(
  	GVL.LS[LS_Mapping.LSHH_204].Status.eStatus=Burkert.DI_Status.Liquid_Detected_Alarm
  	);
  	
  
  //PVl.PID[pid_mapping.Z202_Flow].Actual:=PVL.s8098[s8098_Mapping.FT_203].PDO.VolumeFlow.EU;
  //PV Calculated in Z202-Aux
END_IF;

Z202_Recovery_Level_ctrl(Reverse := true, CV_OK := Network.VFD[vfd_mapping.VFD_202].Ready, PV_OK := PVL.AIT[AIT_Mapping.LT_202].Ready, PID := PVl.PID[pid_mapping.Z202_Recovery_Level ]);
IF Z202_Recovery_Level_ctrl.ENO THEN
  PVl.PID[pid_mapping.Z202_Recovery_Level].InHibit:=(
  	GVL.LS[LS_Mapping.LSHH_204].Status.eStatus=Burkert.DI_Status.Liquid_Detected_Alarm
  	);
  	
  
  PVl.PID[pid_mapping.Z202_Recovery_Level].Actual:=PVL.AIT[AIT_Mapping.LT_202].PCT_Scale;
END_IF;

Z202_Filter_Flow_ctrl(Reverse := False, CV_OK := Network.VFD[vfd_mapping.VFD_202].Ready, PV_OK := PVL.s8098[s8098_Mapping.FT_202].Ready, PID := PVl.PID[pid_mapping.Z202_Filter_Flow ]);
IF Z202_Filter_Flow_ctrl.ENO THEN
  PVl.PID[pid_mapping.Z202_Filter_Flow].InHibit:=(
  	NOT(GVL.Filter_Path_Available) AND 
  	(PVL.Z202_Config.Task.eTask<>eZ202_Task.Drain_P202 AND
  		PVL.Z202_Config.Task.eTask<>eZ202_Task.Drain_P203)
  	);
  	
  
  //PVl.PID[pid_mapping.Z202_Filter_Flow].Actual:=PVL.s8098[s8098_Mapping.FT_202].pdo.VolumeFlow.EU;
  //PV Calculated in Z202-Aux
END_IF;
END_PROGRAM

PROGRAM General_Status_MSG
  VAR
    Local_Status : General_Status;
  END_VAR

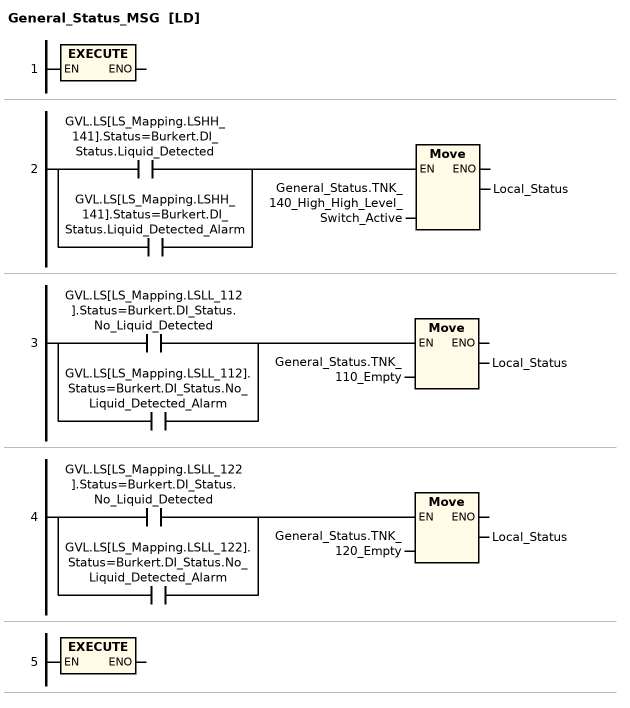
(* LD diagram, written out as Structured Text *)

Local_Status:=General_Status.All_Components_Ready;

IF (GVL.LS[LS_Mapping.LSHH_141].Status=Burkert.DI_Status.Liquid_Detected) OR (GVL.LS[LS_Mapping.LSHH_141].Status=Burkert.DI_Status.Liquid_Detected_Alarm) THEN Local_Status := General_Status.TNK_140_High_High_Level_Switch_Active; END_IF;

IF (GVL.LS[LS_Mapping.LSLL_112 ].Status=Burkert.DI_Status.No_Liquid_Detected) OR (GVL.LS[LS_Mapping.LSLL_112].Status=Burkert.DI_Status.No_Liquid_Detected_Alarm) THEN Local_Status := General_Status.TNK_110_Empty; END_IF;

IF (GVL.LS[LS_Mapping.LSLL_122 ].Status=Burkert.DI_Status.No_Liquid_Detected) OR (GVL.LS[LS_Mapping.LSLL_122].Status=Burkert.DI_Status.No_Liquid_Detected_Alarm) THEN Local_Status := General_Status.TNK_120_Empty; END_IF;




HMI.General_Status:=
	Burkert.Burkert_OSCAT_BASIC.REPLACE_ALL(str:=TO_STRING(Local_Status), src:='_' , rep:=' ' );
END_PROGRAM

PROGRAM RTC_CTRL
  VAR
    stUTC_Timestamp : SysTime;
    stLocal_TimeStamp : SysTime;
    Result : RTS_IEC_RESULT;
    dtNow : DT;
    todNow : TOD;
    datToday : DATE;
    License_Triggered : BOOL;
    Pulse_500ms : Burkert.Burkert_OSCAT_BASIC.clk_PRG;
  END_VAR

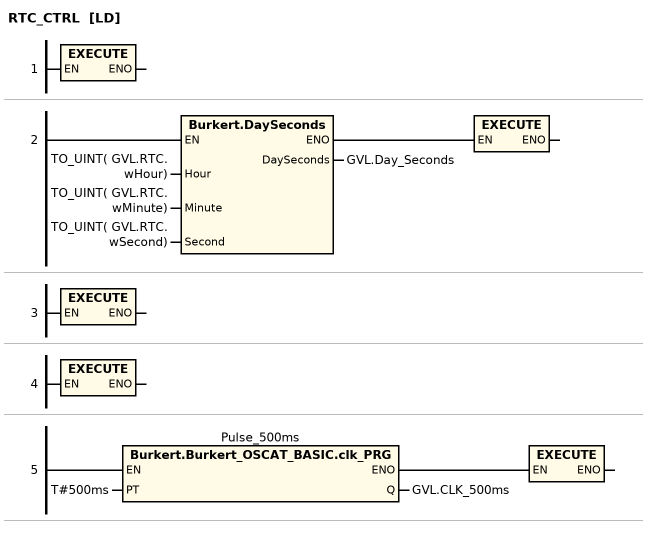
(* LD diagram, written out as Structured Text *)

Result := SysTimeRtcHighResGet(stUTC_Timestamp); // ULINT#1528273494913
Result := SysTimeRtcConvertHighResToLocal(stUTC_Timestamp, GVL.RTC);

// stdNow.wYear = UINT#2018
// stdNow.wMonth = UINT#6
// stdNowy.wDay = UINT#6
// stdNow.wHour = UINT#10
// stdNow.wMinute = UINT#24
// stdNow.wSecond = UINT#54
// stdNow.wMilliseconds = UINT#913
// stdNow.wDayOfWeek = UINT#3
// stdNow.wYday = UINT#157

Result := SysTimeRtcConvertDateToHighRes(GVL.RTC , stLocal_TimeStamp); // ULINT#1528280694913

dtNow := TO_DT(stLocal_TimeStamp / 1000 (* ms *)); // DT#2018-6-6-10:24:54
todNow := TO_TOD(stLocal_TimeStamp MOD TO_ULINT(T#1D)); // TOD#10:24:54.913
datToday := TO_DATE(dtNow); // D#2018-6-6

GVL.Day_Seconds := Burkert.DaySeconds(Hour := TO_UINT( GVL.RTC.wHour), Minute := TO_UINT( GVL.RTC.wMinute), Second := TO_UINT( GVL.RTC.wSecond));
GVL.PLC_Ticker:=GVL.PLC_Ticker+1;
GVL.Local_Epoch:= TO_UDINT(stLocal_TimeStamp MOD TO_ULINT(T#1D));
GVL.UTC_Epoch:= TO_UDINT(stUTC_TimeStamp MOD TO_ULINT(T#1D));

IF
	GVL.RTC.wHour=0	AND
	GVL.RTC.wMinute=5 AND
	GVL.RTC.wSecond=0 
THEN
//
End_IF;

IF (
		(
		PVL.Licence.wYear<> 0 AND
		PVL.Licence.wMonth<>0 AND
		PVL.Licence.wDay<>0 AND
		PVL.Licence.wHour<>0 AND
		PVL.Licence.wMinute<>0 )
		AND 
		(
			GVL.RTC.wYear>=PVL.Licence.wYear AND
			GVL.RTC.wMonth>=PVL.Licence.wMonth	AND
			GVL.RTC.wDay>=PVL.Licence.wDay	AND
			GVL.RTC.wHour>=PVL.Licence.wHour	AND
			GVL.RTC.wMinute>=PVL.Licence.wMinute
		)
	) THEN
	License_Triggered:=TRUE;
		PVL.HMI_Nag:=GVL.RTC.wMinute.3;
	ELSE
		PVL.HMI_Nag:=FALSE;
		License_Triggered:=FALSE;
	END_IF;

Pulse_500ms(PT := T#500ms, Q => GVL.CLK_500ms);
IF Pulse_500ms.ENO THEN
  IF GVL.CLK_500ms THEN
  	GVL.uptime:=GVL.uptime+500;
  END_IF
END_IF;
END_PROGRAM

PROGRAM FIT_Manager
  VAR
    FT_201A_CTRL : Burkert.s8050_UDFB;
    FT_202A_CTRL : Burkert.s8050_UDFB;
    FT_204A_CTRL : Burkert.s8050_UDFB;
    FT_203A_CTRL : Burkert.s8050_UDFB;
  END_VAR

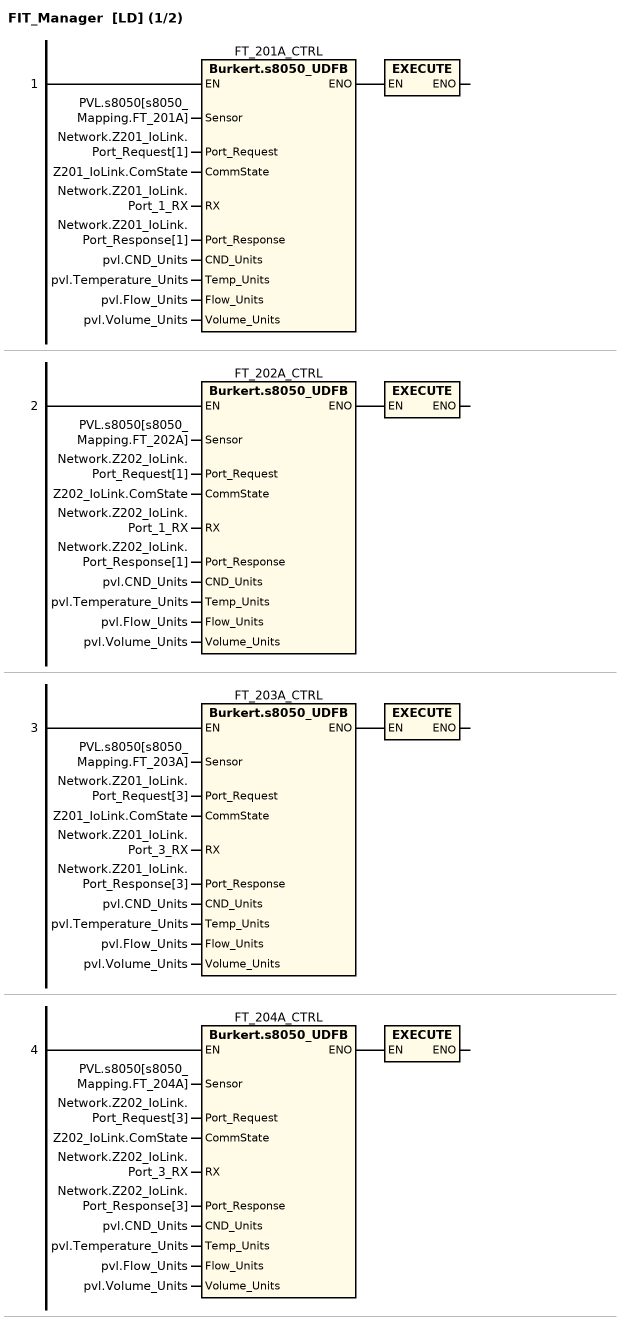
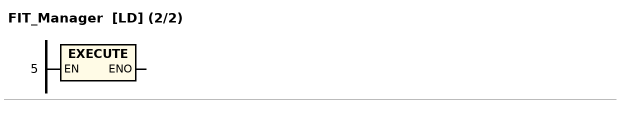
(* LD diagram, written out as Structured Text *)

FT_201A_CTRL(Sensor := PVL.s8050[s8050_Mapping.FT_201A], Port_Request := Network.Z201_IoLink.Port_Request[1], CommState := Z201_IoLink.ComState, RX := Network.Z201_IoLink.Port_1_RX, Port_Response := Network.Z201_IoLink.Port_Response[1], CND_Units := pvl.CND_Units, Temp_Units := pvl.Temperature_Units, Flow_Units := pvl.Flow_Units, Volume_Units := pvl.Volume_Units);
IF FT_201A_CTRL.ENO THEN
  PVL.s8050[s8050_Mapping.FT_201A].CND.Alarm_Config.Silence:=TRUE;
  PVL.s8050[s8050_Mapping.FT_201A].Temp.Alarm_Config.Silence:=TRUE;
  //PVL.s8050[s8050_Mapping.FT_201A].Rate_1.Alarm_Config.Silence:=TRUE;
  
  //PVL.s8050[s8050_Mapping.FT_201A].PLC_Count_Reset:=;
END_IF;

FT_202A_CTRL(Sensor := PVL.s8050[s8050_Mapping.FT_202A], Port_Request := Network.Z202_IoLink.Port_Request[1], CommState := Z202_IoLink.ComState, RX := Network.Z202_IoLink.Port_1_RX, Port_Response := Network.Z202_IoLink.Port_Response[1], CND_Units := pvl.CND_Units, Temp_Units := pvl.Temperature_Units, Flow_Units := pvl.Flow_Units, Volume_Units := pvl.Volume_Units);
IF FT_202A_CTRL.ENO THEN
  PVL.s8050[s8050_Mapping.FT_202A].CND.Alarm_Config.Silence:=TRUE;
  PVL.s8050[s8050_Mapping.FT_202A].Temp.Alarm_Config.Silence:=TRUE;
  //PVL.s8050[s8050_Mapping.FT_202A].Rate_1.Alarm_Config.Silence:=TRUE;
  
  //PVL.s8050[s8050_Mapping.FT_201A].PLC_Count_Reset:=;
END_IF;

FT_203A_CTRL(Sensor := PVL.s8050[s8050_Mapping.FT_203A], Port_Request := Network.Z201_IoLink.Port_Request[3], CommState := Z201_IoLink.ComState, RX := Network.Z201_IoLink.Port_3_RX, Port_Response := Network.Z201_IoLink.Port_Response[3], CND_Units := pvl.CND_Units, Temp_Units := pvl.Temperature_Units, Flow_Units := pvl.Flow_Units, Volume_Units := pvl.Volume_Units);
IF FT_203A_CTRL.ENO THEN
  PVL.s8050[s8050_Mapping.FT_203A].CND.Alarm_Config.Silence:=TRUE;
  PVL.s8050[s8050_Mapping.FT_203A].Temp.Alarm_Config.Silence:=TRUE;
  PVL.s8050[s8050_Mapping.FT_203A].Rate_1.Alarm_Config.Silence:=TRUE;
  
  //PVL.s8050[s8050_Mapping.FT_201A].PLC_Count_Reset:=;
END_IF;

FT_204A_CTRL(Sensor := PVL.s8050[s8050_Mapping.FT_204A], Port_Request := Network.Z202_IoLink.Port_Request[3], CommState := Z202_IoLink.ComState, RX := Network.Z202_IoLink.Port_3_RX, Port_Response := Network.Z202_IoLink.Port_Response[3], CND_Units := pvl.CND_Units, Temp_Units := pvl.Temperature_Units, Flow_Units := pvl.Flow_Units, Volume_Units := pvl.Volume_Units);
IF FT_204A_CTRL.ENO THEN
  PVL.s8050[s8050_Mapping.FT_204A].CND.Alarm_Config.Silence:=TRUE;
  PVL.s8050[s8050_Mapping.FT_204A].Temp.Alarm_Config.Silence:=TRUE;
  //PVL.s8050[s8050_Mapping.FT_204A].Rate_1.Alarm_Config.Silence:=TRUE;
  
  //PVL.s8050[s8050_Mapping.FT_201A].PLC_Count_Reset:=;
END_IF;

PVL.FIT[FIT_Mapping.FT01].Rate.Alarm_Config.Silence:=TRUE;
PVL.fit[fit_mapping.FT01].Total:=Network.ME44_DI[ME44DI_Mapping.GW100_S1].Ch[8].Totaliser;
PVL.fit[fit_mapping.FT01].Rate.EU:=Network.ME44_DI[ME44DI_Mapping.GW100_S1].Ch[8].Hz_Count;
Network.ME44_DI[ME44DI_Mapping.GW100_S1].Ch[8].Reset_Totaliser:=PVL.FIT[FIT_Mapping.FT01].PLC_Reset OR PVL.FIT[FIT_Mapping.FT01].HMI_Reset;
Network.ME44_DI[ME44DI_Mapping.GW100_S1].Ch[8].Reset_Count:=PVL.FIT[FIT_Mapping.FT01].PLC_Reset OR PVL.FIT[FIT_Mapping.FT01].HMI_Reset;

IF PVL.FIT[FIT_Mapping.FT01].HMI_Reset AND PVL.FIT[FIT_Mapping.FT01].Total<0.1 THEN
	PVL.FIT[FIT_Mapping.FT01].HMI_Reset:=FALSE;
END_IF;
END_PROGRAM

PROGRAM s8605_Manager
  VAR
    SV_211_CTRL : Burkert.eDip_8605_CTRL;
    SV_212_CTRL : Burkert.eDip_8605_CTRL;
    SV_217_CTRL : Burkert.eDip_8605_CTRL;
    SV_218_CTRL : Burkert.eDip_8605_CTRL;
    SV_220_CTRL : Burkert.eDip_8605_CTRL;
    SV_221_CTRL : Burkert.eDip_8605_CTRL;
    SV_222_CTRL : Burkert.eDip_8605_CTRL;
    SV_223_CTRL : Burkert.eDip_8605_CTRL;
  END_VAR

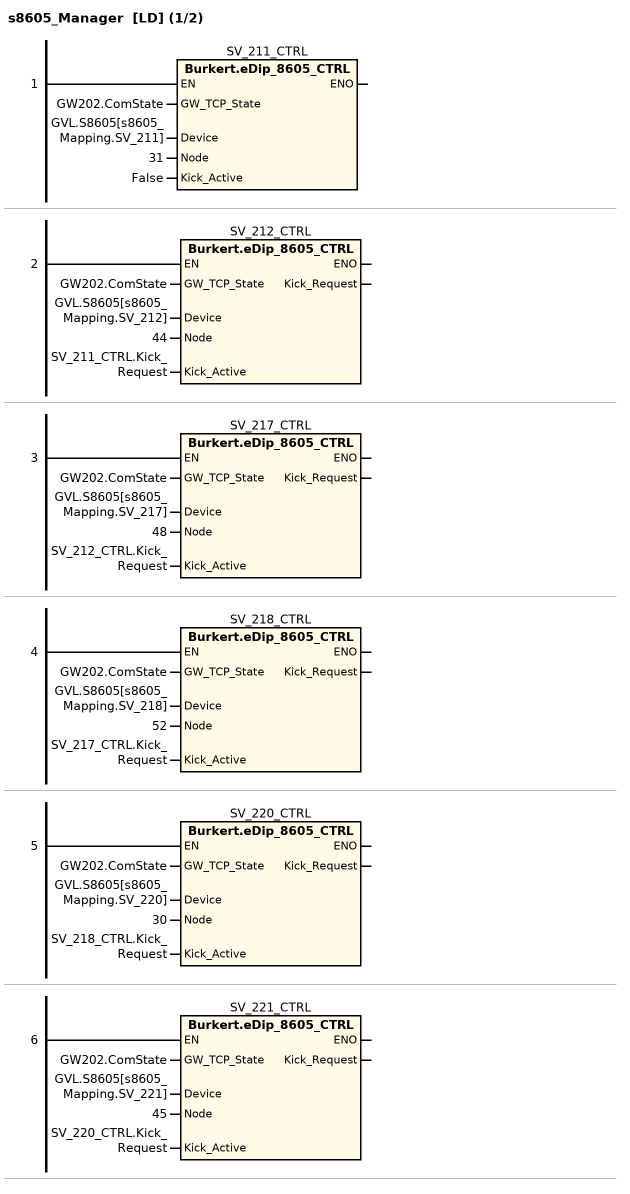
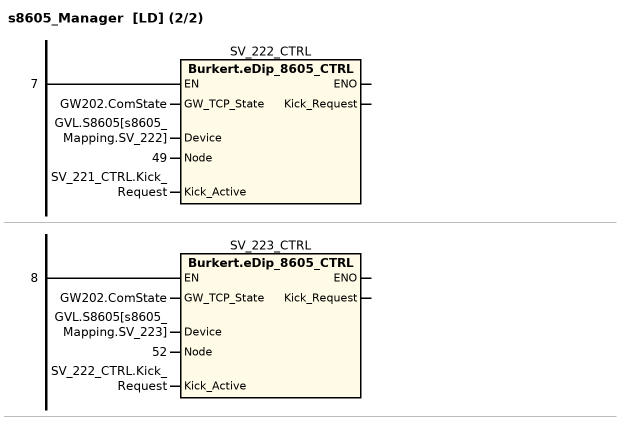
(* LD diagram, written out as Structured Text *)


SV_211_CTRL(GW_TCP_State := GW202.ComState, Device := GVL.S8605[s8605_Mapping.SV_211], Node := 31, Kick_Active := False);

SV_212_CTRL(GW_TCP_State := GW202.ComState, Device := GVL.S8605[s8605_Mapping.SV_212], Node := 44, Kick_Active := SV_211_CTRL.Kick_Request);

SV_217_CTRL(GW_TCP_State := GW202.ComState, Device := GVL.S8605[s8605_Mapping.SV_217], Node := 48, Kick_Active := SV_212_CTRL.Kick_Request);

SV_218_CTRL(GW_TCP_State := GW202.ComState, Device := GVL.S8605[s8605_Mapping.SV_218], Node := 52, Kick_Active := SV_217_CTRL.Kick_Request);

SV_220_CTRL(GW_TCP_State := GW202.ComState, Device := GVL.S8605[s8605_Mapping.SV_220], Node := 30, Kick_Active := SV_218_CTRL.Kick_Request);

SV_221_CTRL(GW_TCP_State := GW202.ComState, Device := GVL.S8605[s8605_Mapping.SV_221], Node := 45, Kick_Active := SV_220_CTRL.Kick_Request);

SV_222_CTRL(GW_TCP_State := GW202.ComState, Device := GVL.S8605[s8605_Mapping.SV_222], Node := 49, Kick_Active := SV_221_CTRL.Kick_Request);

SV_223_CTRL(GW_TCP_State := GW202.ComState, Device := GVL.S8605[s8605_Mapping.SV_223], Node := 52, Kick_Active := SV_222_CTRL.Kick_Request);
END_PROGRAM

PROGRAM HMI_Data
  VAR
    HMI_Contactor : Burkert.Contactor_HMI_Sync_UDFB;
    HMI_Mix : Burkert.Quick_Mix_HMI_Sync_UDFB;
    HMI_Condensate : Burkert.Condensate_HMI_Sync_UDFB;
    HMI_LS : Burkert.DI_HMI_Sync_UDFB;
    HMI_PID : Burkert.PID_HMI_Sync_UDFB;
    HMI_FIT : Burkert.FIT_HMI_Sync_UDFB;
    HMI_AIT : Burkert.AIT_HMI_Sync_UDFB;
    HMI_PT : Burkert.AIT_HMI_Sync_UDFB;
    HMI_TT : Burkert.AIT_HMI_Sync_UDFB;
    HMI_8098 : Burkert.s8098_HMI_Sync_UDFB;
    HMI_Analog_Pump : Burkert.Analog_Pump_HMI_Sync;
    HMI_mPump : Burkert.M_Pump_HMI_Sync;
    HMI_DO : Burkert.DO_HMI_Sync_UDFB;
    HMI_ME64 : Burkert.CanOpen_ME64_HMI_Sync;
    HMI_8228 : Burkert.CanOpen_s8228_HMI_Sync;
    HMI_ACV : Burkert.s336x_HMI_Sync;
    HMI_BCV : Burkert.BCV_HMI_Sync_UDFB;
    HMI_VFD : Burkert.Eaton_VFD_HMI_Sync;  (* HMI_8653: Burkert.CanOpen_8653_HMI_Sync; *)
    HMI_8312 : Burkert.s8312_HMI_Sync;
    HMI_8605 : Burkert.HMI_8605_Sync;
    HMI_8412 : Burkert.s8412_HMI_Sync;
    HMI_8050 : Burkert.s8050_HMI_Sync;
    BCV_Name : BCV_Mapping;
    s336x_Name : s3363_Mapping;
    TT_Name : TT_Mapping;
    PT_Name : s8312_Mapping;
    AIT_Name : AIT_Mapping;
    FIT_Name : FIT_Mapping;
    PID_Name : PID_Mapping;
    LS_Name : LS_Mapping;
    BCV_Name2 : BCV_Mapping;
    SV_Name : SV_Mapping;
    ACV_Name2 : ACV_Mapping;
    VFD_Name : VFD_Mapping;
    s8312_Name : s8312_Mapping;
    s8412_Name : s8412_Mapping;
    s8228_Name : s8228_Mapping;
    s8098_Name : s8098_mapping;
    s8605_Name : s8605_Mapping;
    s8050_Name : s8050_Mapping;
    pump_name : Analog_pump_Mapping;
    mPump_name : mPump_Mapping;
    DO_Name : Do_Mapping;
    ME44AI_Name : ME44AI_Mapping;
  END_VAR
  VAR  (* added by the conversion: wires and edge detectors of the diagram *)
    _Burkert_HMI_ME44AI_Sync187_ENO : BOOL;
    _Burkert_HMI_ME44AI_Sync187_OUT : ANY;
  END_VAR

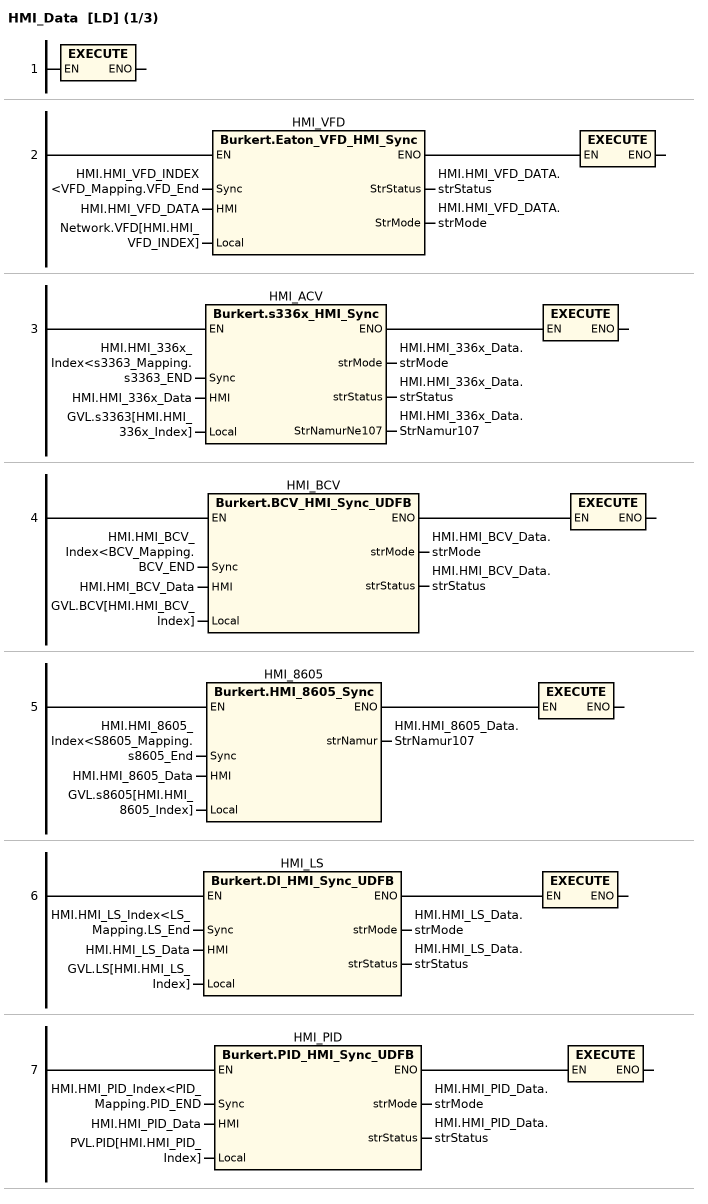
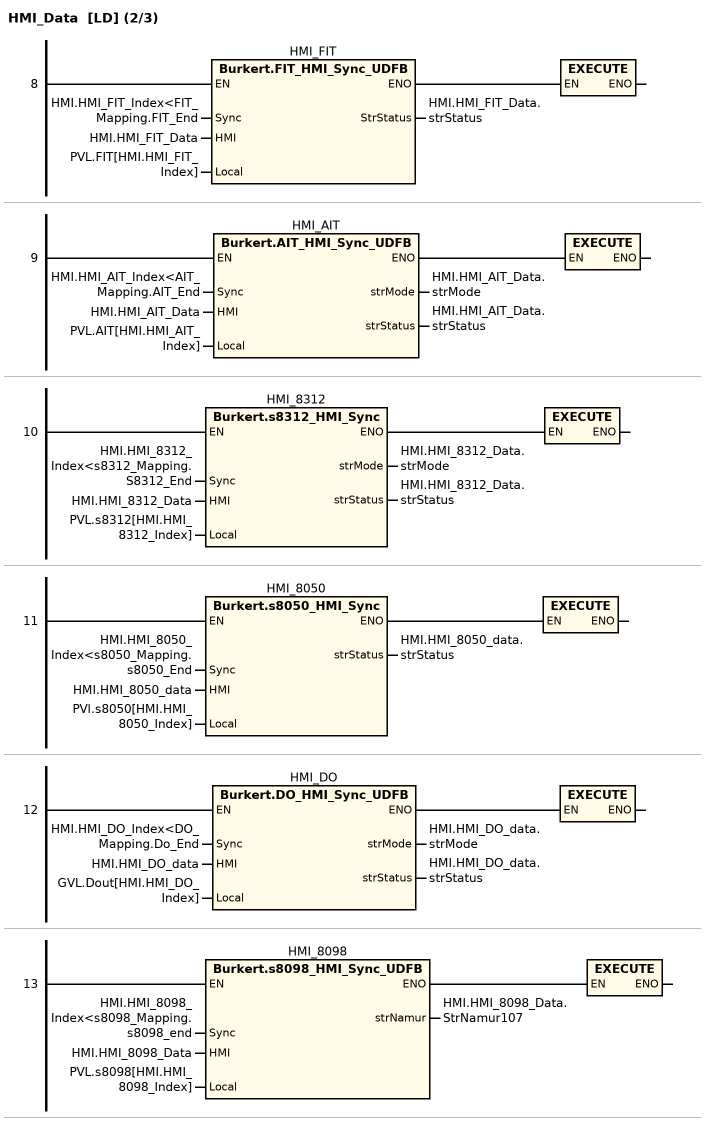
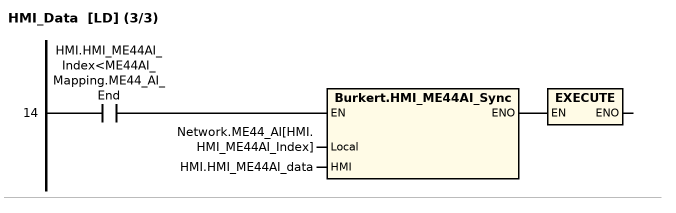
(* LD diagram, written out as Structured Text *)

HMI.StrCND_Units	:=Burkert.Burkert_OSCAT_BASIC.REPLACE_ALL(str:=TO_STRING(PVL.CND_Units) , src:='_' , rep:='/' );
HMI.StrFlow_Units	:=Burkert.Burkert_OSCAT_BASIC.REPLACE_ALL(str:=TO_STRING(PVL.Flow_Units) , src:='_' , rep:='/' );
HMI.StrPressure_Units:=Burkert.Burkert_OSCAT_BASIC.REPLACE_ALL(str:=TO_STRING(PVL.Pressure_Units) , src:='_' , rep:='/' );
HMI.StrResisitivty_Units :=Burkert.Burkert_OSCAT_BASIC.REPLACE_ALL(str:=TO_STRING(PVL.Resisitivty_Units) , src:='_' , rep:='/' );
HMI.StrTDS_Units :=Burkert.Burkert_OSCAT_BASIC.REPLACE_ALL(str:=TO_STRING(PVL.TDS_Units) , src:='_' , rep:='/' );
HMI.StrTemperature_Units :=Burkert.Burkert_OSCAT_BASIC.REPLACE_ALL(str:=TO_STRING(PVL.Temperature_Units) , src:='_' , rep:='/' );
HMI.StrVolume_Units :=Burkert.Burkert_OSCAT_BASIC.REPLACE_ALL(str:=TO_STRING(PVL.Volume_Units) , src:='_' , rep:='/' );

HMI_VFD(Sync := HMI.HMI_VFD_INDEX <VFD_Mapping.VFD_End, HMI := HMI.HMI_VFD_DATA, Local := Network.VFD[HMI.HMI_VFD_INDEX], StrStatus => HMI.HMI_VFD_DATA.strStatus, StrMode => HMI.HMI_VFD_DATA.strMode);
IF HMI_VFD.ENO THEN
  VFD_Name:=HMI.HMI_VFD_Index;
  HMI.HMI_VFD_Data.strName:=Burkert.Burkert_OSCAT_BASIC.REPLACE_ALL(str:=TO_STRING(VFD_Name) , src:='_' , rep:=' ' );
END_IF;

HMI_ACV(Sync := HMI.HMI_336x_Index<s3363_Mapping.s3363_END, HMI := HMI.HMI_336x_Data, Local := GVL.s3363[HMI.HMI_336x_Index], strMode => HMI.HMI_336x_Data.strMode, strStatus => HMI.HMI_336x_Data.strStatus, StrNamurNe107 => HMI.HMI_336x_Data.StrNamur107);
IF HMI_ACV.ENO THEN
  s336x_Name:=HMI.HMI_336x_Index;
  HMI.HMI_336x_Data.strName:=Burkert.Burkert_OSCAT_BASIC.REPLACE_ALL(str:=TO_STRING(s336x_Name) , src:='_' , rep:=' ' );
  HMI.HMI_336x_Data.strTCPstate :=GVL.s3363[HMI.HMI_336x_Index].strTCPstate;
END_IF;

HMI_BCV(Sync := HMI.HMI_BCV_Index<BCV_Mapping.BCV_END, HMI := HMI.HMI_BCV_Data, Local := GVL.BCV[HMI.HMI_BCV_Index], strMode => HMI.HMI_BCV_Data.strMode, strStatus => HMI.HMI_BCV_Data.strStatus);
IF HMI_BCV.ENO THEN
  BCV_Name2:=HMI.HMI_BCV_Index;
  HMI.HMI_BCV_Data.strName:=Burkert.Burkert_OSCAT_BASIC.REPLACE_ALL(str:=TO_STRING(BCV_Name2), src:='_' , rep:=' ' );
END_IF;

HMI_8605(Sync := HMI.HMI_8605_Index<S8605_Mapping.s8605_End, HMI := HMI.HMI_8605_Data, Local := GVL.s8605[HMI.HMI_8605_Index], strNamur => HMI.HMI_8605_Data.StrNamur107);
IF HMI_8605.ENO THEN
  S8605_Name:=HMI.HMI_8605_Index;
  HMI.HMI_8605_Data.strName:=Burkert.Burkert_OSCAT_BASIC.REPLACE_ALL(str:=TO_STRING(S8605_Name), src:='_' , rep:=' ' );
END_IF;

HMI_LS(Sync := HMI.HMI_LS_Index<LS_Mapping.LS_End, HMI := HMI.HMI_LS_Data, Local := GVL.LS[HMI.HMI_LS_Index], strMode => HMI.HMI_LS_Data.strMode, strStatus => HMI.HMI_LS_Data.strStatus);
IF HMI_LS.ENO THEN
  LS_Name:=HMI.HMI_LS_Index;
  HMI.HMI_LS_Data.strName:=Burkert.Burkert_OSCAT_BASIC.REPLACE_ALL(str:=TO_STRING(LS_Name), src:='_' , rep:=' ' );
  //Burkert.Burkert_OSCAT_BASIC.REPLACE_ALL(str:=
  //, src:='_' , rep:=' ' );
END_IF;

HMI_PID(Sync := HMI.HMI_PID_Index<PID_Mapping.PID_END, HMI := HMI.HMI_PID_Data, Local := PVL.PID[HMI.HMI_PID_Index], strMode => HMI.HMI_PID_Data.strMode, strStatus => HMI.HMI_PID_Data.strStatus);
IF HMI_PID.ENO THEN
  PID_Name:=HMI.HMI_PID_Index;
  HMI.HMI_PID_Data.strName:=TO_STRING(PID_Name);
END_IF;

HMI_FIT(Sync := HMI.HMI_FIT_Index<FIT_Mapping.FIT_End, HMI := HMI.HMI_FIT_Data, Local := PVL.FIT[HMI.HMI_FIT_Index], StrStatus => HMI.HMI_FIT_Data.strStatus);
IF HMI_FIT.ENO THEN
  FIT_Name:=HMI.HMI_FIT_Index;
  HMI.HMI_FIT_Data.strName:=Burkert.Burkert_OSCAT_BASIC.REPLACE_ALL(str:=TO_STRING(FIT_Name), src:='_' , rep:=' ' );
END_IF;

HMI_AIT(Sync := HMI.HMI_AIT_Index<AIT_Mapping.AIT_End, HMI := HMI.HMI_AIT_Data, Local := PVL.AIT[HMI.HMI_AIT_Index], strMode => HMI.HMI_AIT_Data.strMode, strStatus => HMI.HMI_AIT_Data.strStatus);
IF HMI_AIT.ENO THEN
  AIT_Name:=HMI.HMI_AIT_Index;
  HMI.HMI_AIT_Data.strName:=TO_STRING(AIT_Name);
END_IF;

HMI_8312(Sync := HMI.HMI_8312_Index<s8312_Mapping.S8312_End, HMI := HMI.HMI_8312_Data, Local := PVL.s8312[HMI.HMI_8312_Index], strMode => HMI.HMI_8312_Data.strMode, strStatus => HMI.HMI_8312_Data.strStatus);
IF HMI_8312.ENO THEN
  s8312_Name:=HMI.HMI_8312_Index;
  HMI.HMI_8312_Data.strName:=Burkert.Burkert_OSCAT_BASIC.REPLACE_ALL(str:=TO_STRING(s8312_Name) , src:='_' , rep:=' ' );
END_IF;

HMI_8050(Sync := HMI.HMI_8050_Index<s8050_Mapping.s8050_End, HMI := HMI.HMI_8050_data, Local := PVl.s8050[HMI.HMI_8050_Index], strStatus => HMI.HMI_8050_data.strStatus);
IF HMI_8050.ENO THEN
  s8050_name:=HMI.HMI_8050_Index;
  HMI.HMI_8050_data.strName:=TO_STRING(S8050_Name);
END_IF;

